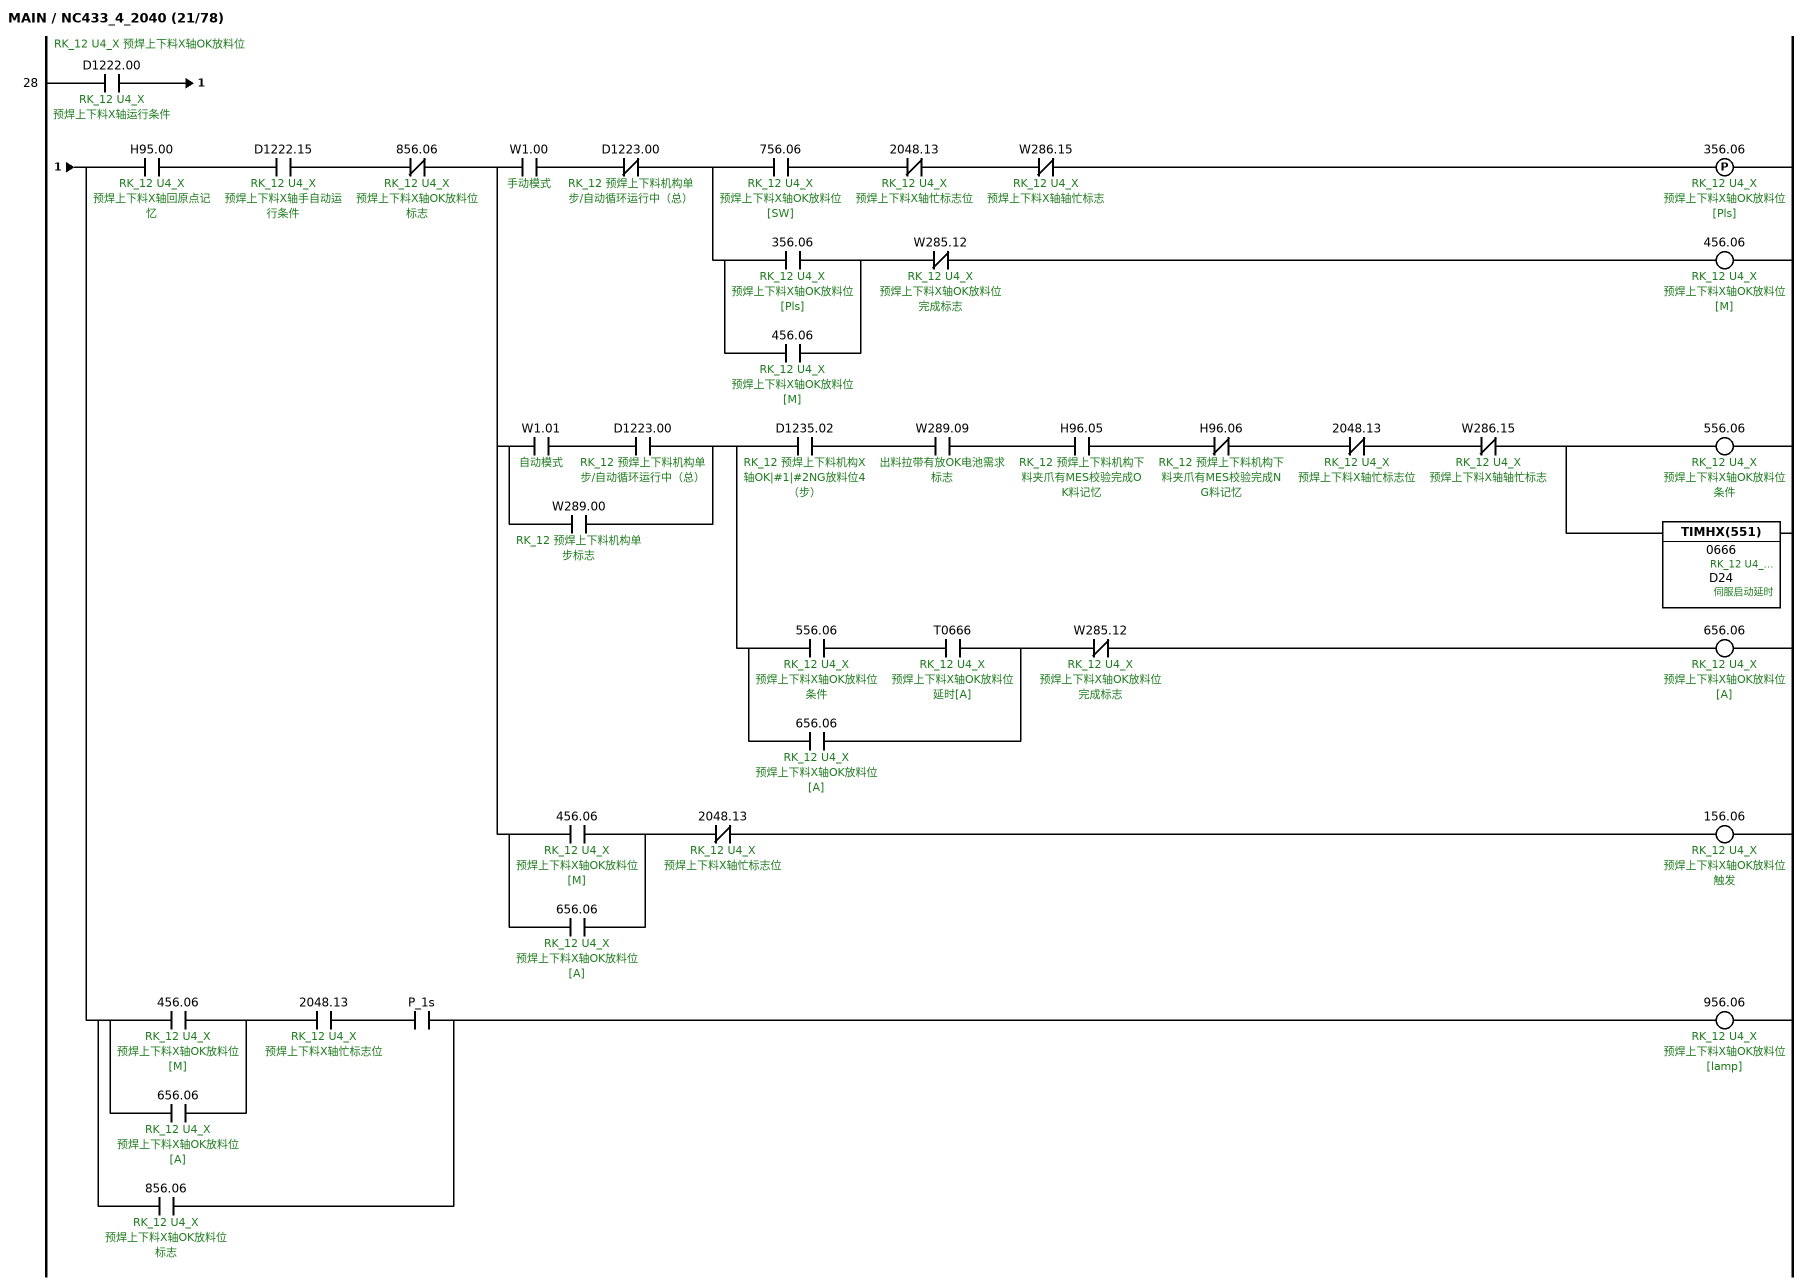
; [picture p168: MAIN / NC433_4_2040, rungs 28-28]
; rung 28: RK_12 U4_X 预焊上下料X轴OK放料位
LD D1222.00  ; RK_12 U4_X 预焊上下料X轴运行条件
OUT TR0
AND H95.00  ; RK_12 U4_X 预焊上下料X轴回原点记忆
AND D1222.15  ; RK_12 U4_X 预焊上下料X轴手自动运行条件
ANDNOT 856.06  ; RK_12 U4_X 预焊上下料X轴OK放料位标志
OUT TR1
AND W1.00  ; 手动模式
ANDNOT D1223.00  ; RK_12 预焊上下料机构单步/自动循环运行中（总）
OUT TR2
AND 756.06  ; RK_12 U4_X 预焊上下料X轴OK放料位[SW]
ANDNOT 2048.13  ; RK_12 U4_X 预焊上下料X轴忙标志位
ANDNOT W286.15  ; RK_12 U4_X 预焊上下料X轴轴忙标志
DIFU(013) 356.06  ; RK_12 U4_X 预焊上下料X轴OK放料位[Pls]
LD TR2
LD 356.06  ; RK_12 U4_X 预焊上下料X轴OK放料位[Pls]
OR 456.06  ; RK_12 U4_X 预焊上下料X轴OK放料位[M]
ANDLD
ANDNOT W285.12  ; RK_12 U4_X 预焊上下料X轴OK放料位完成标志
OUT 456.06  ; RK_12 U4_X 预焊上下料X轴OK放料位[M]
LD TR1
LD W1.01  ; 自动模式
AND D1223.00  ; RK_12 预焊上下料机构单步/自动循环运行中（总）
OR W289.00  ; RK_12 预焊上下料机构单步标志
ANDLD
OUT TR2
AND D1235.02  ; RK_12 预焊上下料机构X轴OK|#1|#2NG放料位4（步）
AND W289.09  ; 出料拉带有放OK电池需求标志
AND H96.05  ; RK_12 预焊上下料机构下料夹爪有MES校验完成OK料记忆
ANDNOT H96.06  ; RK_12 预焊上下料机构下料夹爪有MES校验完成NG料记忆
ANDNOT 2048.13  ; RK_12 U4_X 预焊上下料X轴忙标志位
ANDNOT W286.15  ; RK_12 U4_X 预焊上下料X轴轴忙标志
OUT 556.06  ; RK_12 U4_X 预焊上下料X轴OK放料位条件
TIMHX(551) 0666 D24  ; 伺服启动延时, RK_12 U4_X 预焊上下料X轴OK放料位延时[A]
LD TR2
LD 556.06  ; RK_12 U4_X 预焊上下料X轴OK放料位条件
AND T0666  ; RK_12 U4_X 预焊上下料X轴OK放料位延时[A]
OR 656.06  ; RK_12 U4_X 预焊上下料X轴OK放料位[A]
ANDLD
ANDNOT W285.12  ; RK_12 U4_X 预焊上下料X轴OK放料位完成标志
OUT 656.06  ; RK_12 U4_X 预焊上下料X轴OK放料位[A]
LD TR1
LD 456.06  ; RK_12 U4_X 预焊上下料X轴OK放料位[M]
OR 656.06  ; RK_12 U4_X 预焊上下料X轴OK放料位[A]
ANDLD
ANDNOT 2048.13  ; RK_12 U4_X 预焊上下料X轴忙标志位
OUT 156.06  ; RK_12 U4_X 预焊上下料X轴OK放料位触发
LD TR0
LD 456.06  ; RK_12 U4_X 预焊上下料X轴OK放料位[M]
OR 656.06  ; RK_12 U4_X 预焊上下料X轴OK放料位[A]
AND 2048.13  ; RK_12 U4_X 预焊上下料X轴忙标志位
AND P_1s
OR 856.06  ; RK_12 U4_X 预焊上下料X轴OK放料位标志
ANDLD
OUT 956.06  ; RK_12 U4_X 预焊上下料X轴OK放料位[lamp]

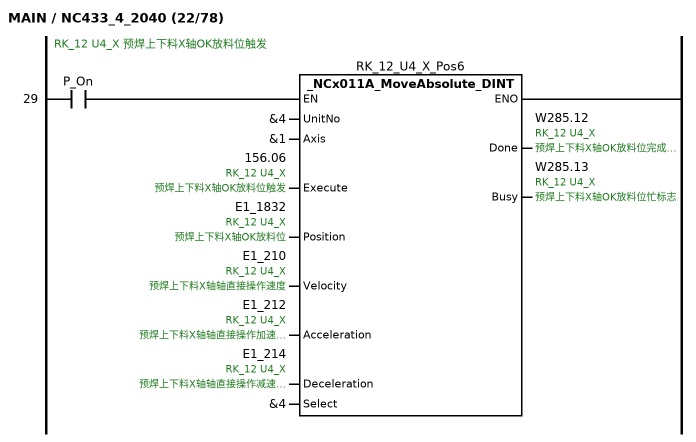
; rung 29: RK_12 U4_X 预焊上下料X轴OK放料位触发
LD P_On
CALL RK_12_U4_X_Pos6 : _NCx011A_MoveAbsolute_DINT (UnitNo := &4, Axis := &1, Execute := 156.06, Position := E1_1832, Velocity := E1_210, Acceleration := E1_212, Deceleration := E1_214, Select := &4, Done => W285.12, Busy => W285.13)  ; RK_12 U4_X 预焊上下料X轴OK放料位触发, RK_12 U4_X 预焊上下料X轴OK放料位, RK_12 U4_X 预焊上下料X轴轴直接操作速度, RK_12 U4_X 预焊上下料X轴轴直接操作加速时间, RK_12 U4_X 预焊上下料X轴轴直接操作减速时间, RK_12 U4_X 预焊上下料X轴OK放料位完成标志, RK_12 U4_X 预焊上下料X轴OK放料位忙标志

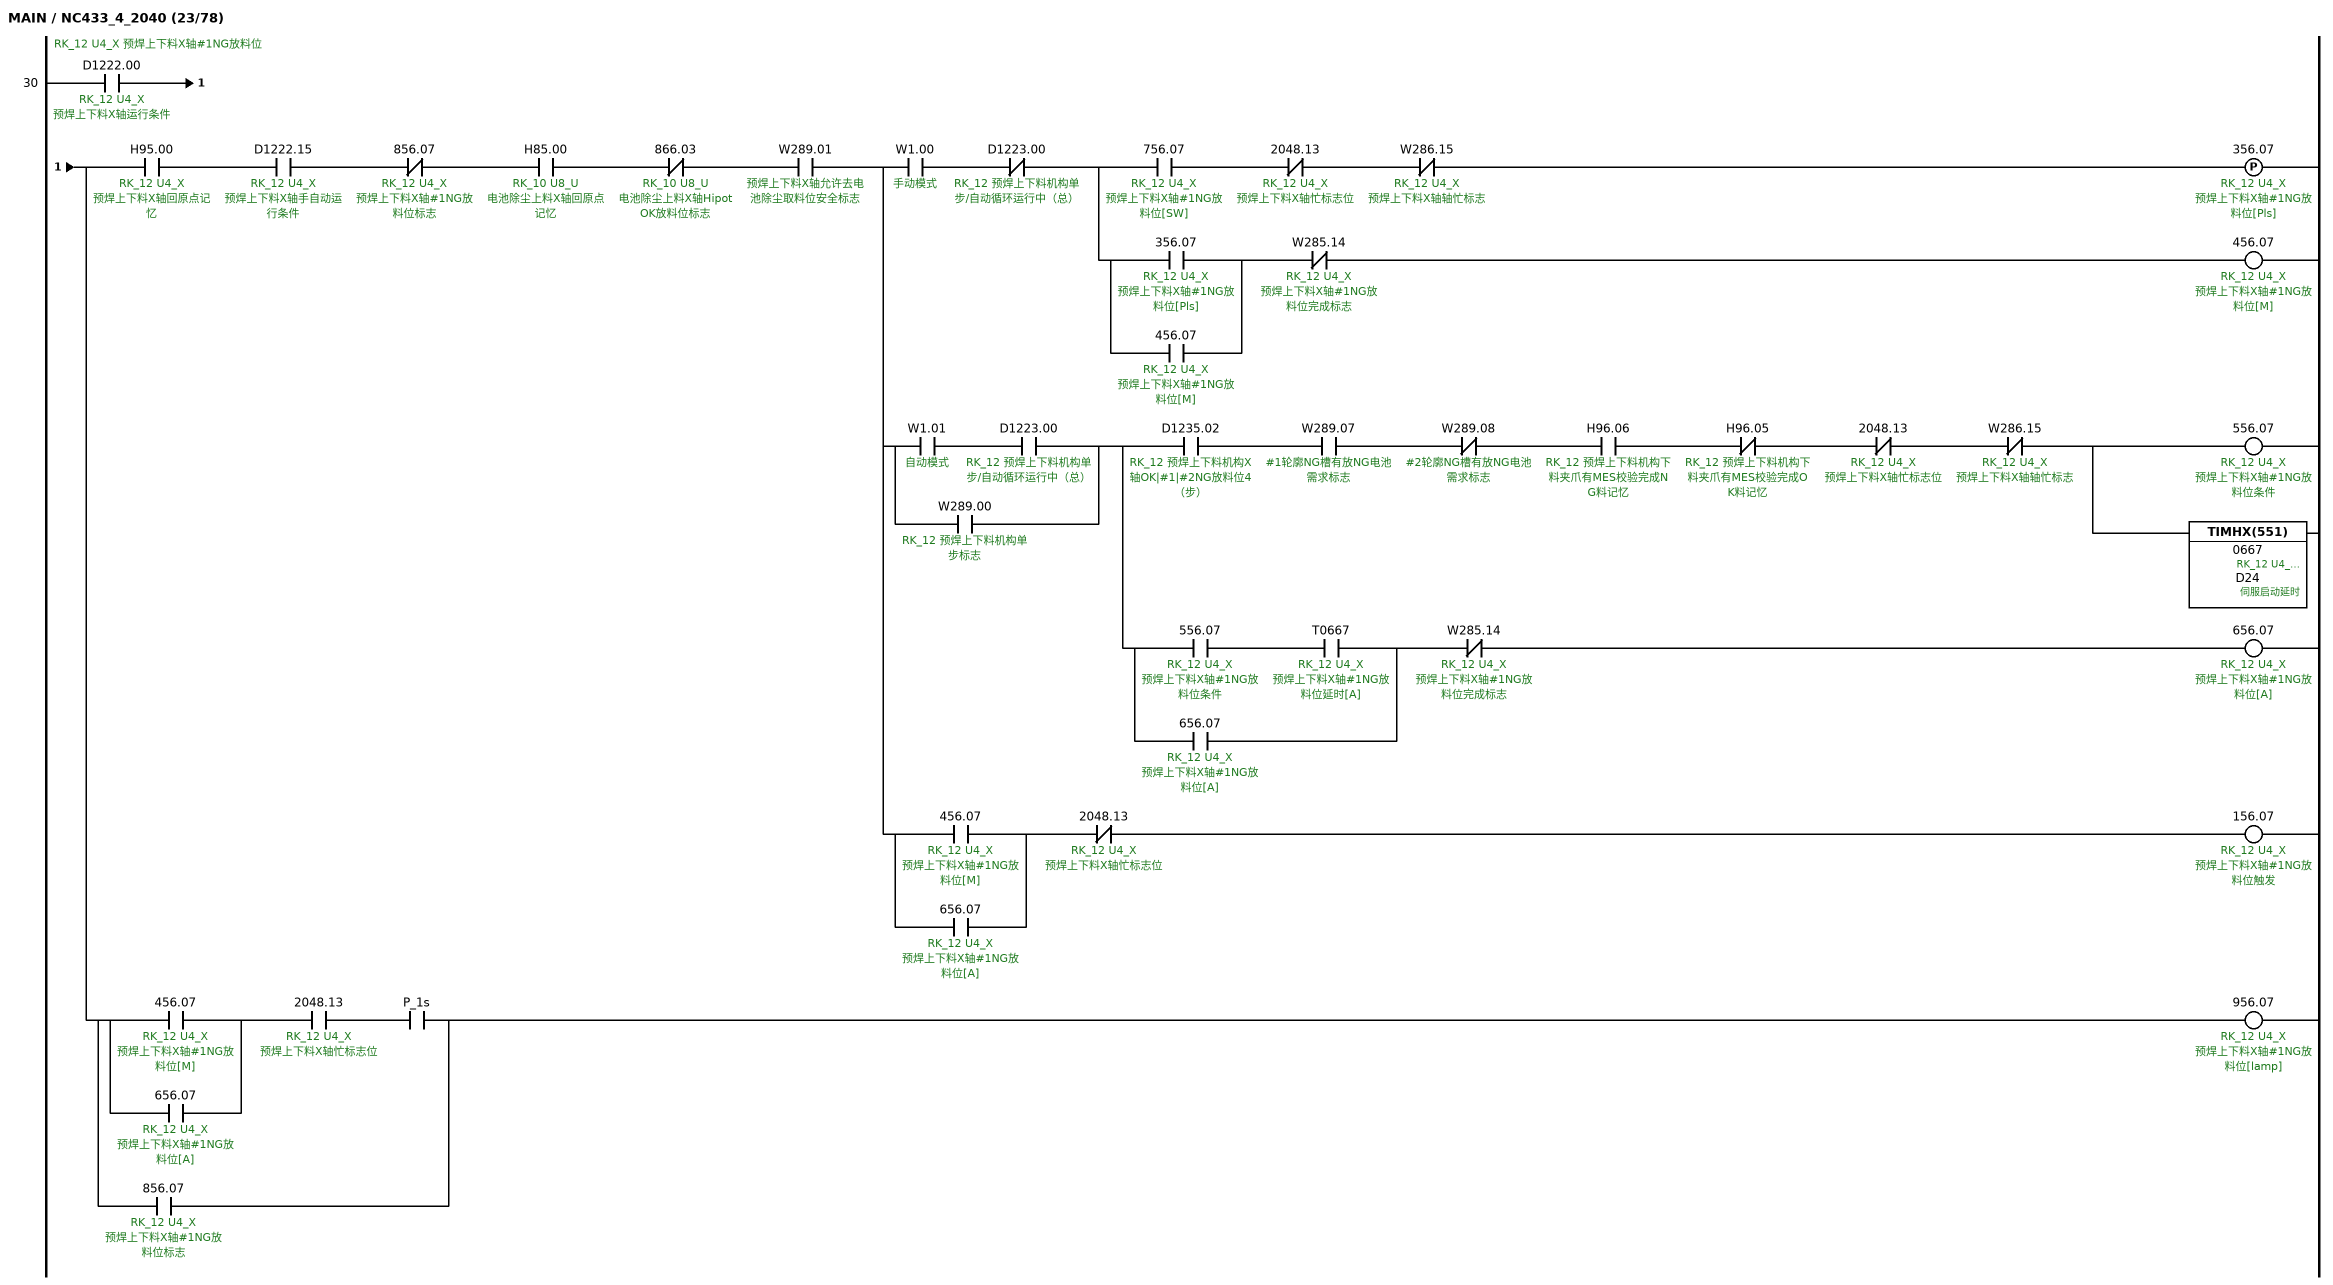
; rung 30: RK_12 U4_X 预焊上下料X轴#1NG放料位
LD D1222.00  ; RK_12 U4_X 预焊上下料X轴运行条件
OUT TR0
AND H95.00  ; RK_12 U4_X 预焊上下料X轴回原点记忆
AND D1222.15  ; RK_12 U4_X 预焊上下料X轴手自动运行条件
ANDNOT 856.07  ; RK_12 U4_X 预焊上下料X轴#1NG放料位标志
AND H85.00  ; RK_10 U8_U 电池除尘上料X轴回原点记忆
ANDNOT 866.03  ; RK_10 U8_U 电池除尘上料X轴Hipot OK放料位标志
AND W289.01  ; 预焊上下料X轴允许去电池除尘取料位安全标志
OUT TR1
AND W1.00  ; 手动模式
ANDNOT D1223.00  ; RK_12 预焊上下料机构单步/自动循环运行中（总）
OUT TR2
AND 756.07  ; RK_12 U4_X 预焊上下料X轴#1NG放料位[SW]
ANDNOT 2048.13  ; RK_12 U4_X 预焊上下料X轴忙标志位
ANDNOT W286.15  ; RK_12 U4_X 预焊上下料X轴轴忙标志
DIFU(013) 356.07  ; RK_12 U4_X 预焊上下料X轴#1NG放料位[Pls]
LD TR2
LD 356.07  ; RK_12 U4_X 预焊上下料X轴#1NG放料位[Pls]
OR 456.07  ; RK_12 U4_X 预焊上下料X轴#1NG放料位[M]
ANDLD
ANDNOT W285.14  ; RK_12 U4_X 预焊上下料X轴#1NG放料位完成标志
OUT 456.07  ; RK_12 U4_X 预焊上下料X轴#1NG放料位[M]
LD TR1
LD W1.01  ; 自动模式
AND D1223.00  ; RK_12 预焊上下料机构单步/自动循环运行中（总）
OR W289.00  ; RK_12 预焊上下料机构单步标志
ANDLD
OUT TR2
AND D1235.02  ; RK_12 预焊上下料机构X轴OK|#1|#2NG放料位4（步）
AND W289.07  ; #1轮廓NG槽有放NG电池需求标志
ANDNOT W289.08  ; #2轮廓NG槽有放NG电池需求标志
AND H96.06  ; RK_12 预焊上下料机构下料夹爪有MES校验完成NG料记忆
ANDNOT H96.05  ; RK_12 预焊上下料机构下料夹爪有MES校验完成OK料记忆
ANDNOT 2048.13  ; RK_12 U4_X 预焊上下料X轴忙标志位
ANDNOT W286.15  ; RK_12 U4_X 预焊上下料X轴轴忙标志
OUT 556.07  ; RK_12 U4_X 预焊上下料X轴#1NG放料位条件
TIMHX(551) 0667 D24  ; 伺服启动延时, RK_12 U4_X 预焊上下料X轴#1NG放料位延时[A]
LD TR2
LD 556.07  ; RK_12 U4_X 预焊上下料X轴#1NG放料位条件
AND T0667  ; RK_12 U4_X 预焊上下料X轴#1NG放料位延时[A]
OR 656.07  ; RK_12 U4_X 预焊上下料X轴#1NG放料位[A]
ANDLD
ANDNOT W285.14  ; RK_12 U4_X 预焊上下料X轴#1NG放料位完成标志
OUT 656.07  ; RK_12 U4_X 预焊上下料X轴#1NG放料位[A]
LD TR1
LD 456.07  ; RK_12 U4_X 预焊上下料X轴#1NG放料位[M]
OR 656.07  ; RK_12 U4_X 预焊上下料X轴#1NG放料位[A]
ANDLD
ANDNOT 2048.13  ; RK_12 U4_X 预焊上下料X轴忙标志位
OUT 156.07  ; RK_12 U4_X 预焊上下料X轴#1NG放料位触发
LD TR0
LD 456.07  ; RK_12 U4_X 预焊上下料X轴#1NG放料位[M]
OR 656.07  ; RK_12 U4_X 预焊上下料X轴#1NG放料位[A]
AND 2048.13  ; RK_12 U4_X 预焊上下料X轴忙标志位
AND P_1s
OR 856.07  ; RK_12 U4_X 预焊上下料X轴#1NG放料位标志
ANDLD
OUT 956.07  ; RK_12 U4_X 预焊上下料X轴#1NG放料位[lamp]

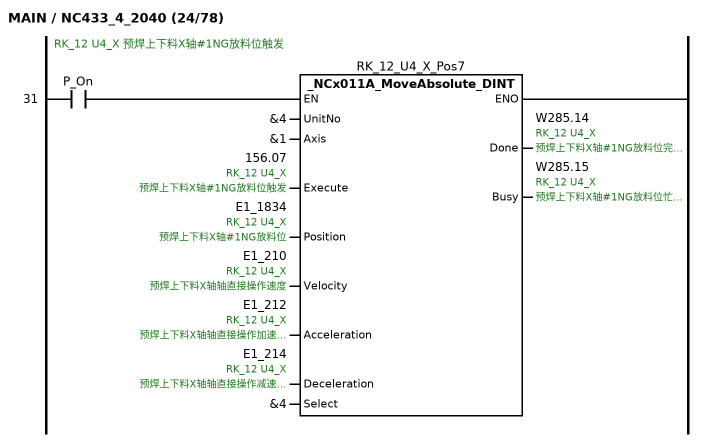
; rung 31: RK_12 U4_X 预焊上下料X轴#1NG放料位触发
LD P_On
CALL RK_12_U4_X_Pos7 : _NCx011A_MoveAbsolute_DINT (UnitNo := &4, Axis := &1, Execute := 156.07, Position := E1_1834, Velocity := E1_210, Acceleration := E1_212, Deceleration := E1_214, Select := &4, Done => W285.14, Busy => W285.15)  ; RK_12 U4_X 预焊上下料X轴#1NG放料位触发, RK_12 U4_X 预焊上下料X轴#1NG放料位, RK_12 U4_X 预焊上下料X轴轴直接操作速度, RK_12 U4_X 预焊上下料X轴轴直接操作加速时间, RK_12 U4_X 预焊上下料X轴轴直接操作减速时间, RK_12 U4_X 预焊上下料X轴#1NG放料位完成标志, RK_12 U4_X 预焊上下料X轴#1NG放料位忙标志

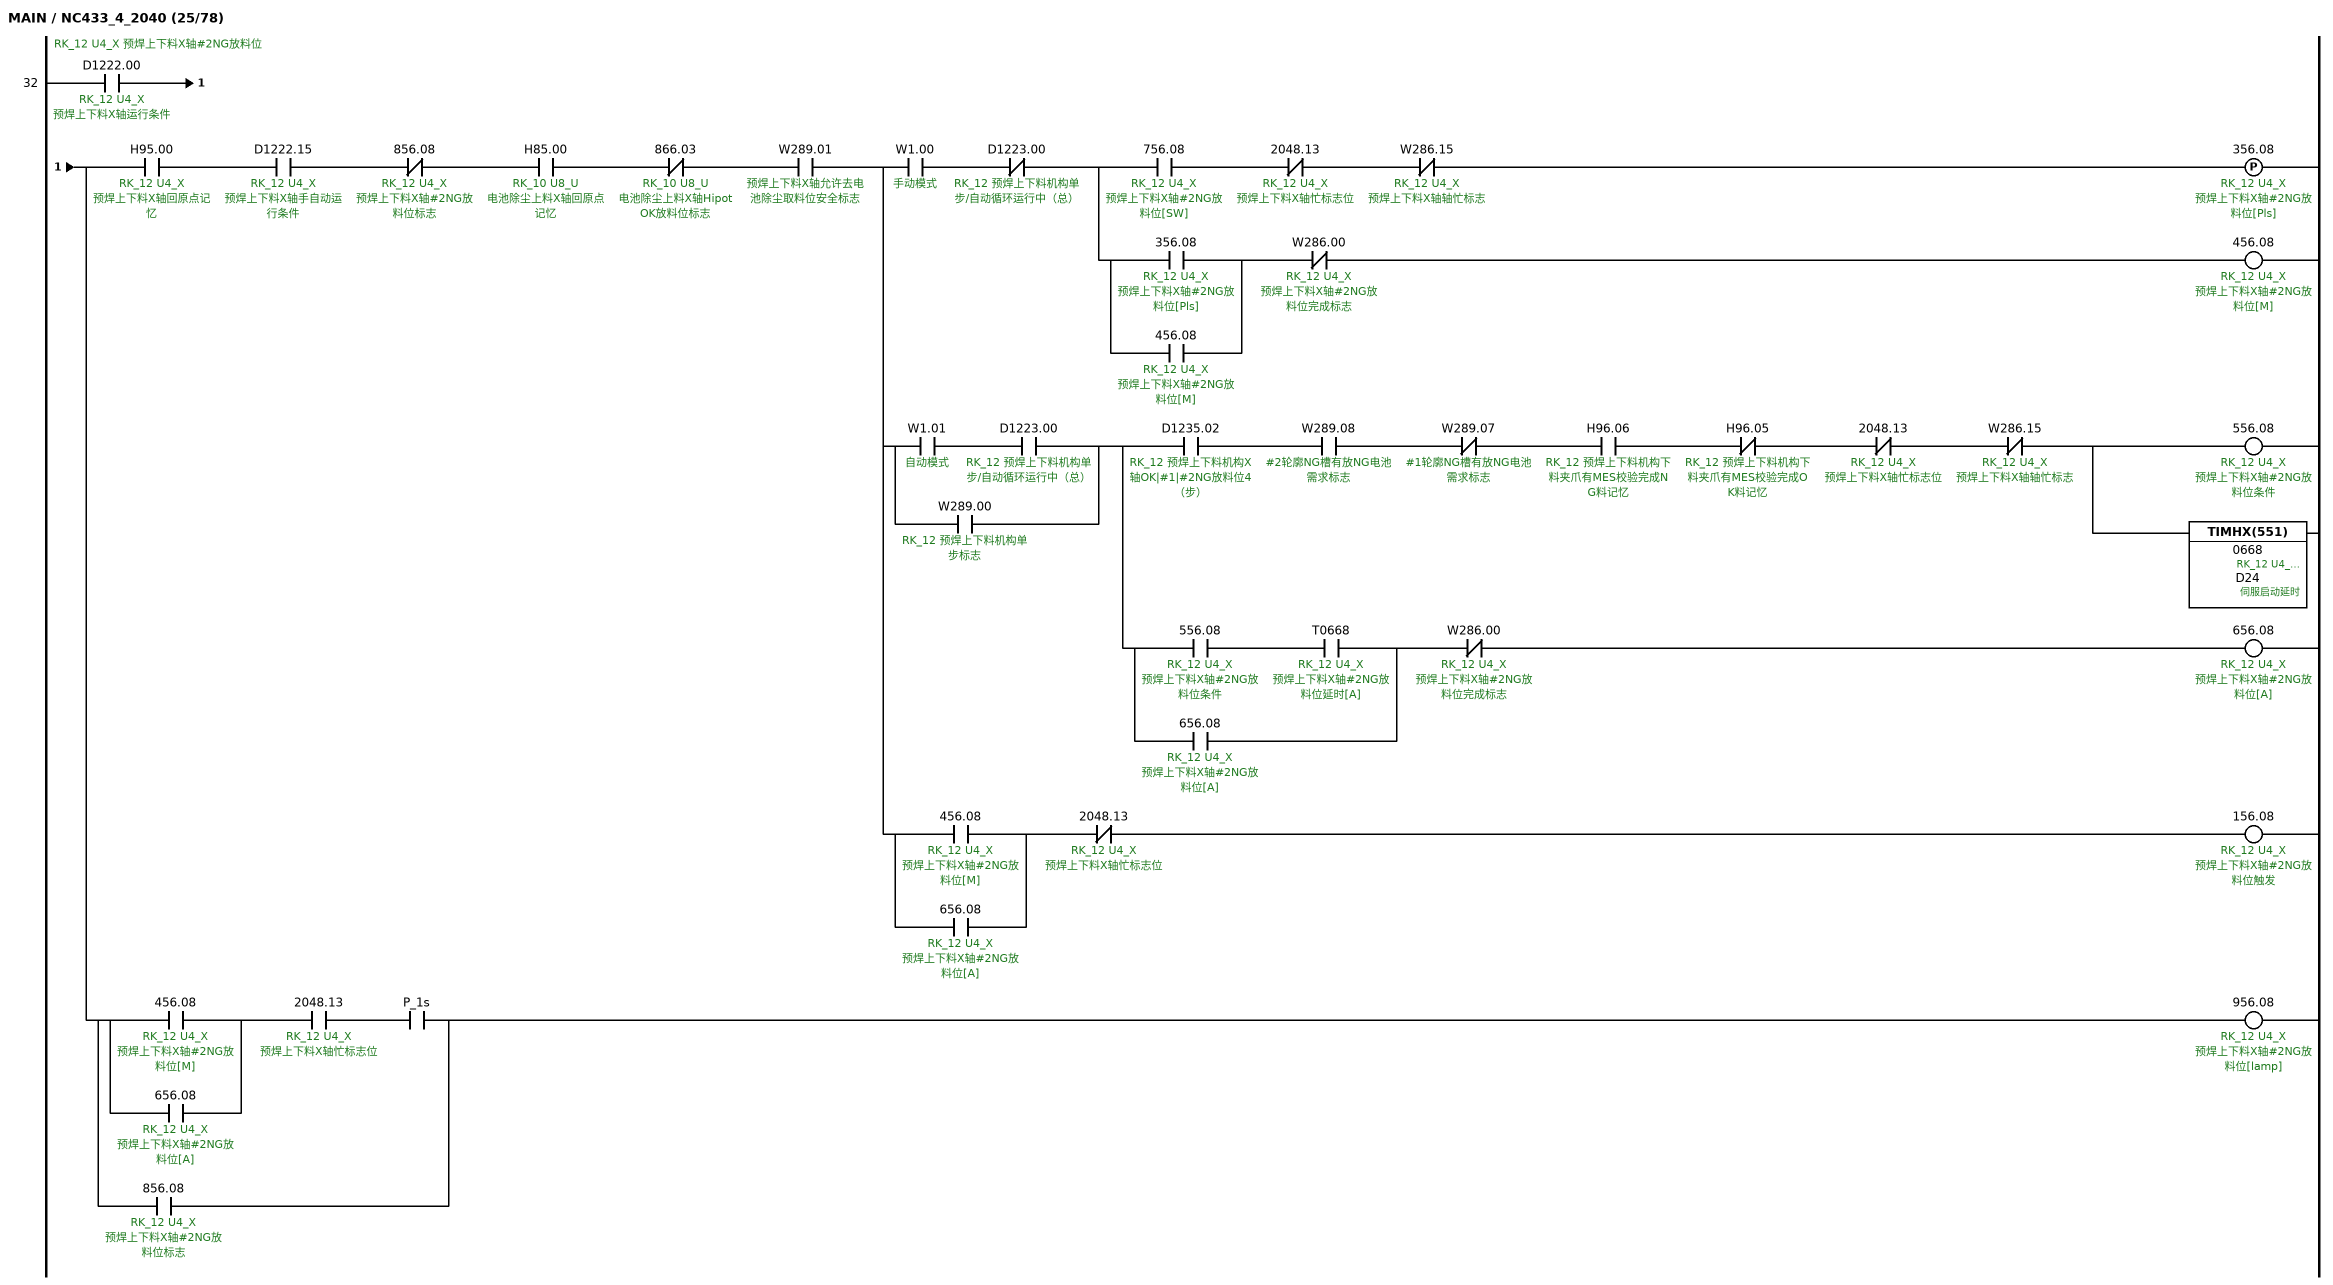
; rung 32: RK_12 U4_X 预焊上下料X轴#2NG放料位
LD D1222.00  ; RK_12 U4_X 预焊上下料X轴运行条件
OUT TR0
AND H95.00  ; RK_12 U4_X 预焊上下料X轴回原点记忆
AND D1222.15  ; RK_12 U4_X 预焊上下料X轴手自动运行条件
ANDNOT 856.08  ; RK_12 U4_X 预焊上下料X轴#2NG放料位标志
AND H85.00  ; RK_10 U8_U 电池除尘上料X轴回原点记忆
ANDNOT 866.03  ; RK_10 U8_U 电池除尘上料X轴Hipot OK放料位标志
AND W289.01  ; 预焊上下料X轴允许去电池除尘取料位安全标志
OUT TR1
AND W1.00  ; 手动模式
ANDNOT D1223.00  ; RK_12 预焊上下料机构单步/自动循环运行中（总）
OUT TR2
AND 756.08  ; RK_12 U4_X 预焊上下料X轴#2NG放料位[SW]
ANDNOT 2048.13  ; RK_12 U4_X 预焊上下料X轴忙标志位
ANDNOT W286.15  ; RK_12 U4_X 预焊上下料X轴轴忙标志
DIFU(013) 356.08  ; RK_12 U4_X 预焊上下料X轴#2NG放料位[Pls]
LD TR2
LD 356.08  ; RK_12 U4_X 预焊上下料X轴#2NG放料位[Pls]
OR 456.08  ; RK_12 U4_X 预焊上下料X轴#2NG放料位[M]
ANDLD
ANDNOT W286.00  ; RK_12 U4_X 预焊上下料X轴#2NG放料位完成标志
OUT 456.08  ; RK_12 U4_X 预焊上下料X轴#2NG放料位[M]
LD TR1
LD W1.01  ; 自动模式
AND D1223.00  ; RK_12 预焊上下料机构单步/自动循环运行中（总）
OR W289.00  ; RK_12 预焊上下料机构单步标志
ANDLD
OUT TR2
AND D1235.02  ; RK_12 预焊上下料机构X轴OK|#1|#2NG放料位4（步）
AND W289.08  ; #2轮廓NG槽有放NG电池需求标志
ANDNOT W289.07  ; #1轮廓NG槽有放NG电池需求标志
AND H96.06  ; RK_12 预焊上下料机构下料夹爪有MES校验完成NG料记忆
ANDNOT H96.05  ; RK_12 预焊上下料机构下料夹爪有MES校验完成OK料记忆
ANDNOT 2048.13  ; RK_12 U4_X 预焊上下料X轴忙标志位
ANDNOT W286.15  ; RK_12 U4_X 预焊上下料X轴轴忙标志
OUT 556.08  ; RK_12 U4_X 预焊上下料X轴#2NG放料位条件
TIMHX(551) 0668 D24  ; 伺服启动延时, RK_12 U4_X 预焊上下料X轴#2NG放料位延时[A]
LD TR2
LD 556.08  ; RK_12 U4_X 预焊上下料X轴#2NG放料位条件
AND T0668  ; RK_12 U4_X 预焊上下料X轴#2NG放料位延时[A]
OR 656.08  ; RK_12 U4_X 预焊上下料X轴#2NG放料位[A]
ANDLD
ANDNOT W286.00  ; RK_12 U4_X 预焊上下料X轴#2NG放料位完成标志
OUT 656.08  ; RK_12 U4_X 预焊上下料X轴#2NG放料位[A]
LD TR1
LD 456.08  ; RK_12 U4_X 预焊上下料X轴#2NG放料位[M]
OR 656.08  ; RK_12 U4_X 预焊上下料X轴#2NG放料位[A]
ANDLD
ANDNOT 2048.13  ; RK_12 U4_X 预焊上下料X轴忙标志位
OUT 156.08  ; RK_12 U4_X 预焊上下料X轴#2NG放料位触发
LD TR0
LD 456.08  ; RK_12 U4_X 预焊上下料X轴#2NG放料位[M]
OR 656.08  ; RK_12 U4_X 预焊上下料X轴#2NG放料位[A]
AND 2048.13  ; RK_12 U4_X 预焊上下料X轴忙标志位
AND P_1s
OR 856.08  ; RK_12 U4_X 预焊上下料X轴#2NG放料位标志
ANDLD
OUT 956.08  ; RK_12 U4_X 预焊上下料X轴#2NG放料位[lamp]

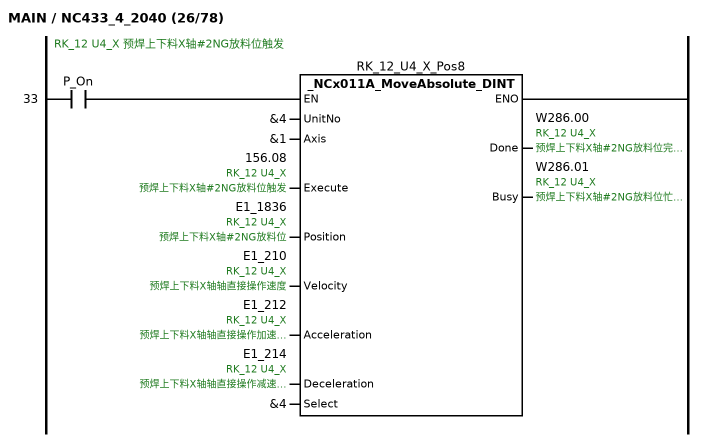
; rung 33: RK_12 U4_X 预焊上下料X轴#2NG放料位触发
LD P_On
CALL RK_12_U4_X_Pos8 : _NCx011A_MoveAbsolute_DINT (UnitNo := &4, Axis := &1, Execute := 156.08, Position := E1_1836, Velocity := E1_210, Acceleration := E1_212, Deceleration := E1_214, Select := &4, Done => W286.00, Busy => W286.01)  ; RK_12 U4_X 预焊上下料X轴#2NG放料位触发, RK_12 U4_X 预焊上下料X轴#2NG放料位, RK_12 U4_X 预焊上下料X轴轴直接操作速度, RK_12 U4_X 预焊上下料X轴轴直接操作加速时间, RK_12 U4_X 预焊上下料X轴轴直接操作减速时间, RK_12 U4_X 预焊上下料X轴#2NG放料位完成标志, RK_12 U4_X 预焊上下料X轴#2NG放料位忙标志

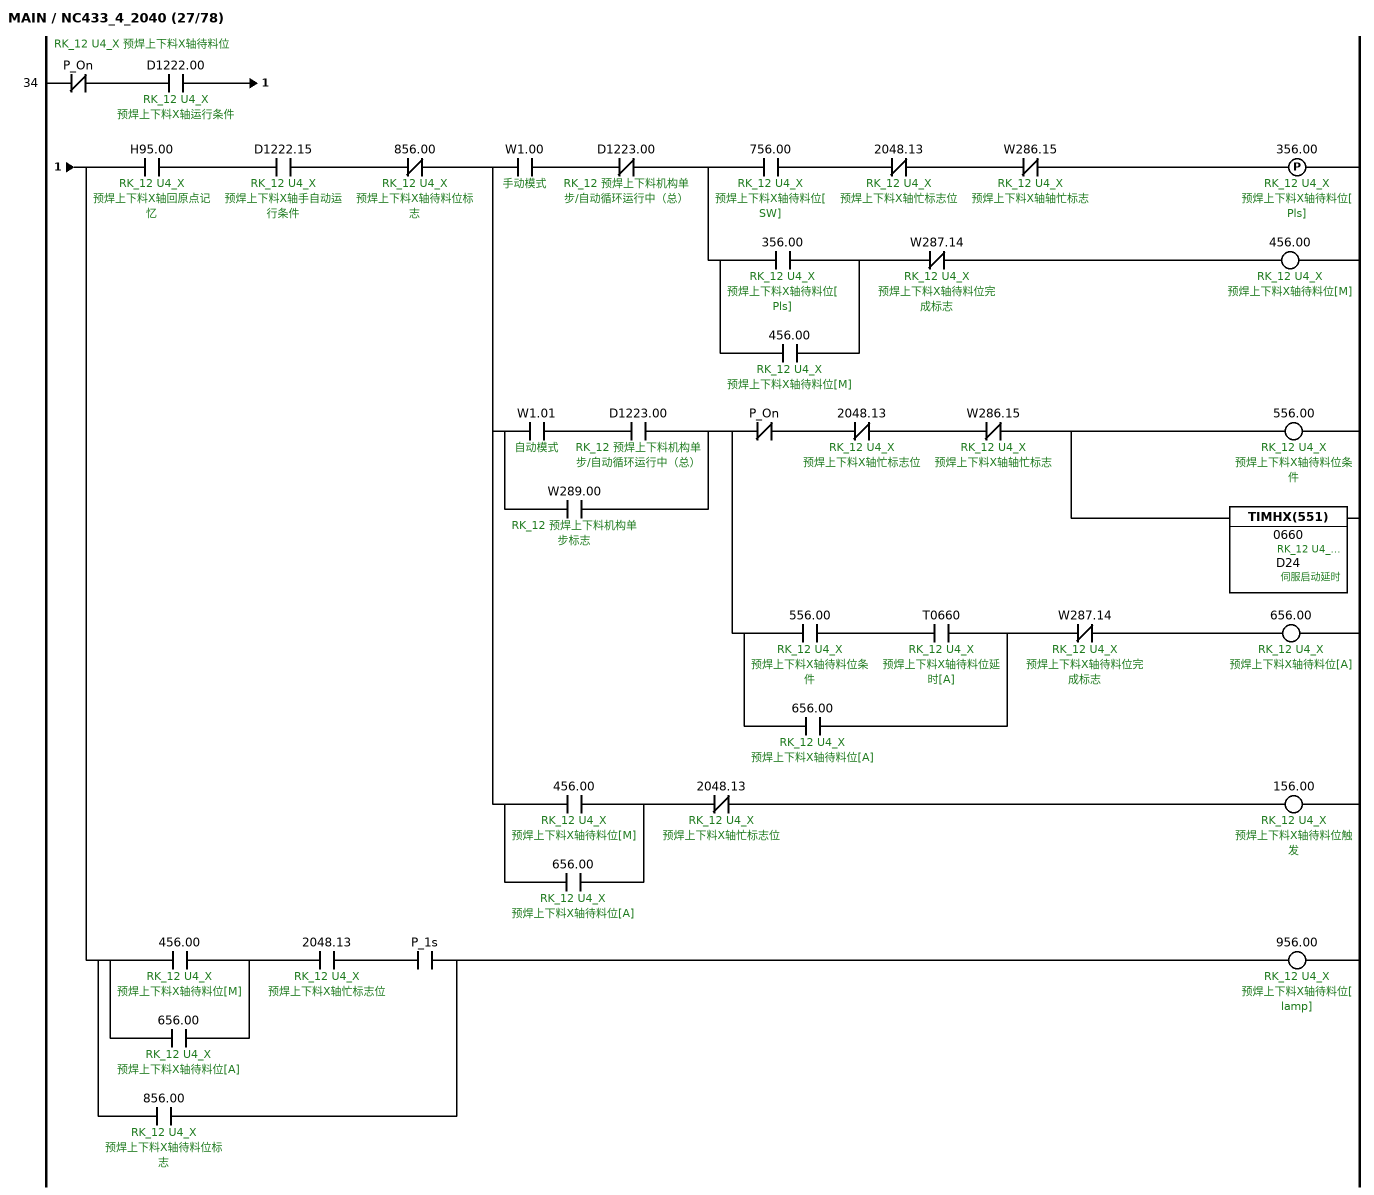
; rung 34: RK_12 U4_X 预焊上下料X轴待料位
LDNOT P_On
AND D1222.00  ; RK_12 U4_X 预焊上下料X轴运行条件
OUT TR0
AND H95.00  ; RK_12 U4_X 预焊上下料X轴回原点记忆
AND D1222.15  ; RK_12 U4_X 预焊上下料X轴手自动运行条件
ANDNOT 856.00  ; RK_12 U4_X 预焊上下料X轴待料位标志
OUT TR1
AND W1.00  ; 手动模式
ANDNOT D1223.00  ; RK_12 预焊上下料机构单步/自动循环运行中（总）
OUT TR2
AND 756.00  ; RK_12 U4_X 预焊上下料X轴待料位[SW]
ANDNOT 2048.13  ; RK_12 U4_X 预焊上下料X轴忙标志位
ANDNOT W286.15  ; RK_12 U4_X 预焊上下料X轴轴忙标志
DIFU(013) 356.00  ; RK_12 U4_X 预焊上下料X轴待料位[Pls]
LD TR2
LD 356.00  ; RK_12 U4_X 预焊上下料X轴待料位[Pls]
OR 456.00  ; RK_12 U4_X 预焊上下料X轴待料位[M]
ANDLD
ANDNOT W287.14  ; RK_12 U4_X 预焊上下料X轴待料位完成标志
OUT 456.00  ; RK_12 U4_X 预焊上下料X轴待料位[M]
LD TR1
LD W1.01  ; 自动模式
AND D1223.00  ; RK_12 预焊上下料机构单步/自动循环运行中（总）
OR W289.00  ; RK_12 预焊上下料机构单步标志
ANDLD
OUT TR2
ANDNOT P_On  // RK_12 U4_X 预焊上下料X轴待料位（步）
ANDNOT 2048.13  ; RK_12 U4_X 预焊上下料X轴忙标志位
ANDNOT W286.15  ; RK_12 U4_X 预焊上下料X轴轴忙标志
OUT 556.00  ; RK_12 U4_X 预焊上下料X轴待料位条件
TIMHX(551) 0660 D24  ; 伺服启动延时, RK_12 U4_X 预焊上下料X轴待料位延时[A]
LD TR2
LD 556.00  ; RK_12 U4_X 预焊上下料X轴待料位条件
AND T0660  ; RK_12 U4_X 预焊上下料X轴待料位延时[A]
OR 656.00  ; RK_12 U4_X 预焊上下料X轴待料位[A]
ANDLD
ANDNOT W287.14  ; RK_12 U4_X 预焊上下料X轴待料位完成标志
OUT 656.00  ; RK_12 U4_X 预焊上下料X轴待料位[A]
LD TR1
LD 456.00  ; RK_12 U4_X 预焊上下料X轴待料位[M]
OR 656.00  ; RK_12 U4_X 预焊上下料X轴待料位[A]
ANDLD
ANDNOT 2048.13  ; RK_12 U4_X 预焊上下料X轴忙标志位
OUT 156.00  ; RK_12 U4_X 预焊上下料X轴待料位触发
LD TR0
LD 456.00  ; RK_12 U4_X 预焊上下料X轴待料位[M]
OR 656.00  ; RK_12 U4_X 预焊上下料X轴待料位[A]
AND 2048.13  ; RK_12 U4_X 预焊上下料X轴忙标志位
AND P_1s
OR 856.00  ; RK_12 U4_X 预焊上下料X轴待料位标志
ANDLD
OUT 956.00  ; RK_12 U4_X 预焊上下料X轴待料位[lamp]

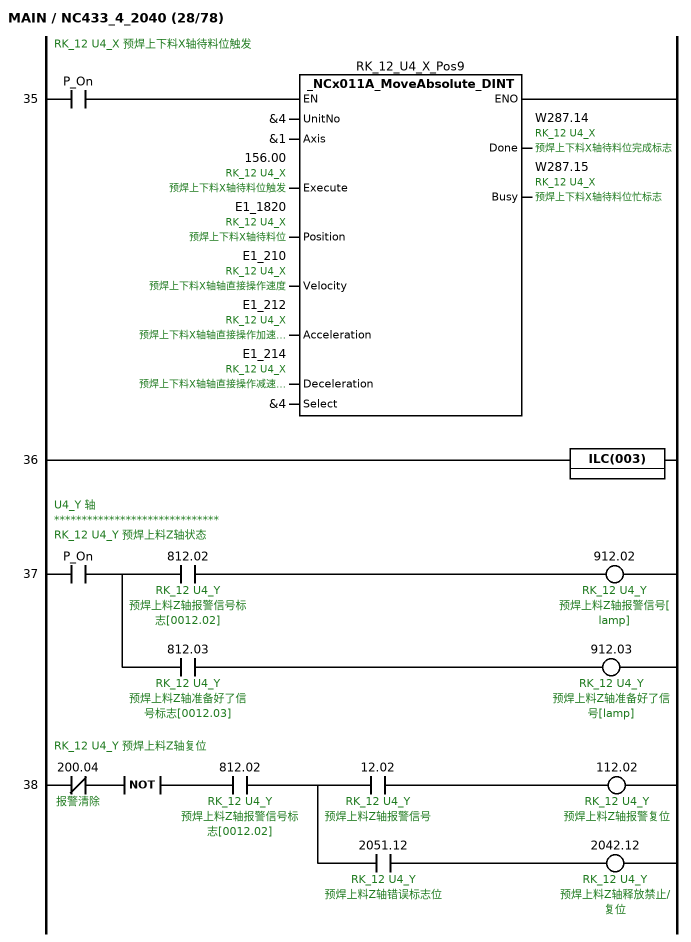
; rung 35: RK_12 U4_X 预焊上下料X轴待料位触发
LD P_On
CALL RK_12_U4_X_Pos9 : _NCx011A_MoveAbsolute_DINT (UnitNo := &4, Axis := &1, Execute := 156.00, Position := E1_1820, Velocity := E1_210, Acceleration := E1_212, Deceleration := E1_214, Select := &4, Done => W287.14, Busy => W287.15)  ; RK_12 U4_X 预焊上下料X轴待料位触发, RK_12 U4_X 预焊上下料X轴待料位, RK_12 U4_X 预焊上下料X轴轴直接操作速度, RK_12 U4_X 预焊上下料X轴轴直接操作加速时间, RK_12 U4_X 预焊上下料X轴轴直接操作减速时间, RK_12 U4_X 预焊上下料X轴待料位完成标志, RK_12 U4_X 预焊上下料X轴待料位忙标志
; rung 36
ILC(003)
; rung 37: U4_Y 轴 / ****************************** / RK_12 U4_Y 预焊上料Z轴状态
LD P_On
OUT TR0
AND 812.02  ; RK_12 U4_Y 预焊上料Z轴报警信号标志[0012.02]
OUT 912.02  ; RK_12 U4_Y 预焊上料Z轴报警信号[lamp]
LD TR0
AND 812.03  ; RK_12 U4_Y 预焊上料Z轴准备好了信号标志[0012.03]
OUT 912.03  ; RK_12 U4_Y 预焊上料Z轴准备好了信号[lamp]
; rung 38: RK_12 U4_Y 预焊上料Z轴复位
LDNOT 200.04  ; 报警清除
NOT(520)
AND 812.02  ; RK_12 U4_Y 预焊上料Z轴报警信号标志[0012.02]
OUT TR0
AND 12.02  ; RK_12 U4_Y 预焊上料Z轴报警信号
OUT 112.02  ; RK_12 U4_Y 预焊上料Z轴报警复位
LD TR0
AND 2051.12  ; RK_12 U4_Y 预焊上料Z轴错误标志位
OUT 2042.12  ; RK_12 U4_Y 预焊上料Z轴释放禁止/复位

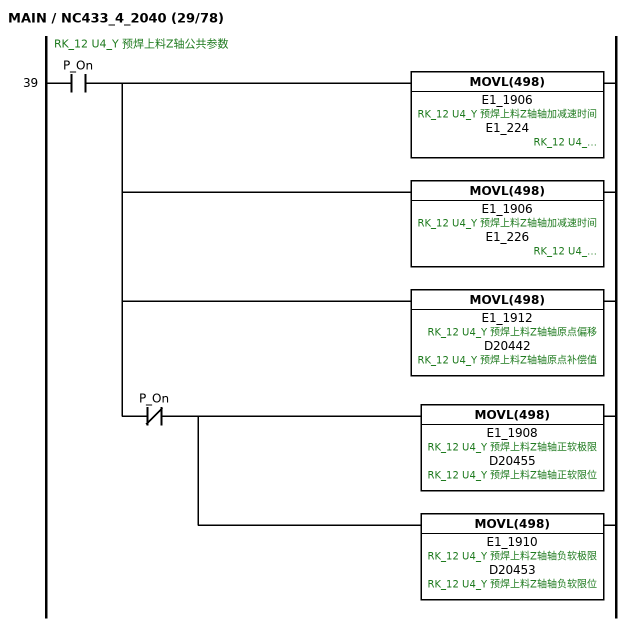
; rung 39: RK_12 U4_Y 预焊上料Z轴公共参数
LD P_On
MOVL(498) E1_1906 E1_224  ; RK_12 U4_Y 预焊上料Z轴轴加减速时间, RK_12 U4_Y 预焊上料Z轴轴直接操作加速时间
MOVL(498) E1_1906 E1_226  ; RK_12 U4_Y 预焊上料Z轴轴加减速时间, RK_12 U4_Y 预焊上料Z轴轴直接操作减速时间
MOVL(498) E1_1912 D20442  ; RK_12 U4_Y 预焊上料Z轴轴原点偏移, RK_12 U4_Y 预焊上料Z轴轴原点补偿值
ANDNOT P_On
MOVL(498) E1_1908 D20455  ; RK_12 U4_Y 预焊上料Z轴轴正软极限, RK_12 U4_Y 预焊上料Z轴轴正软限位
MOVL(498) E1_1910 D20453  ; RK_12 U4_Y 预焊上料Z轴轴负软极限, RK_12 U4_Y 预焊上料Z轴轴负软限位

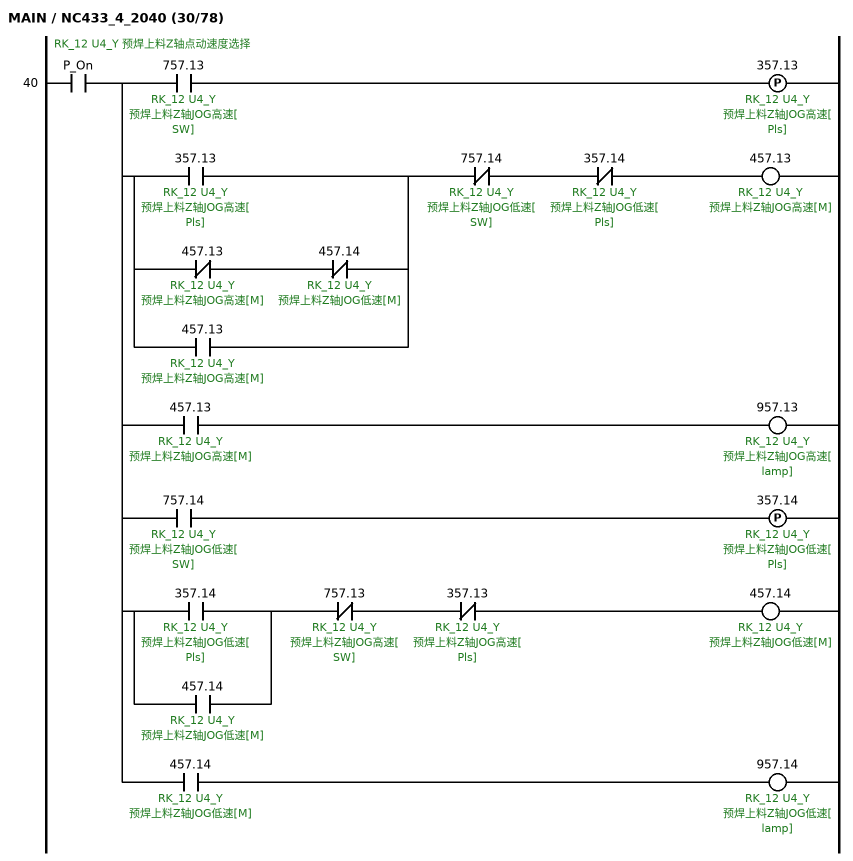
; rung 40: RK_12 U4_Y 预焊上料Z轴点动速度选择
LD P_On
OUT TR0
AND 757.13  ; RK_12 U4_Y 预焊上料Z轴JOG高速[SW]
DIFU(013) 357.13  ; RK_12 U4_Y 预焊上料Z轴JOG高速[Pls]
LD TR0
LD 357.13  ; RK_12 U4_Y 预焊上料Z轴JOG高速[Pls]
LDNOT 457.13  ; RK_12 U4_Y 预焊上料Z轴JOG高速[M]
ANDNOT 457.14  ; RK_12 U4_Y 预焊上料Z轴JOG低速[M]
ORLD
OR 457.13  ; RK_12 U4_Y 预焊上料Z轴JOG高速[M]
ANDLD
ANDNOT 757.14  ; RK_12 U4_Y 预焊上料Z轴JOG低速[SW]
ANDNOT 357.14  ; RK_12 U4_Y 预焊上料Z轴JOG低速[Pls]
OUT 457.13  ; RK_12 U4_Y 预焊上料Z轴JOG高速[M]
LD TR0
AND 457.13  ; RK_12 U4_Y 预焊上料Z轴JOG高速[M]
OUT 957.13  ; RK_12 U4_Y 预焊上料Z轴JOG高速[lamp]
LD TR0
AND 757.14  ; RK_12 U4_Y 预焊上料Z轴JOG低速[SW]
DIFU(013) 357.14  ; RK_12 U4_Y 预焊上料Z轴JOG低速[Pls]
LD TR0
LD 357.14  ; RK_12 U4_Y 预焊上料Z轴JOG低速[Pls]
OR 457.14  ; RK_12 U4_Y 预焊上料Z轴JOG低速[M]
ANDLD
ANDNOT 757.13  ; RK_12 U4_Y 预焊上料Z轴JOG高速[SW]
ANDNOT 357.13  ; RK_12 U4_Y 预焊上料Z轴JOG高速[Pls]
OUT 457.14  ; RK_12 U4_Y 预焊上料Z轴JOG低速[M]
LD TR0
AND 457.14  ; RK_12 U4_Y 预焊上料Z轴JOG低速[M]
OUT 957.14  ; RK_12 U4_Y 预焊上料Z轴JOG低速[lamp]

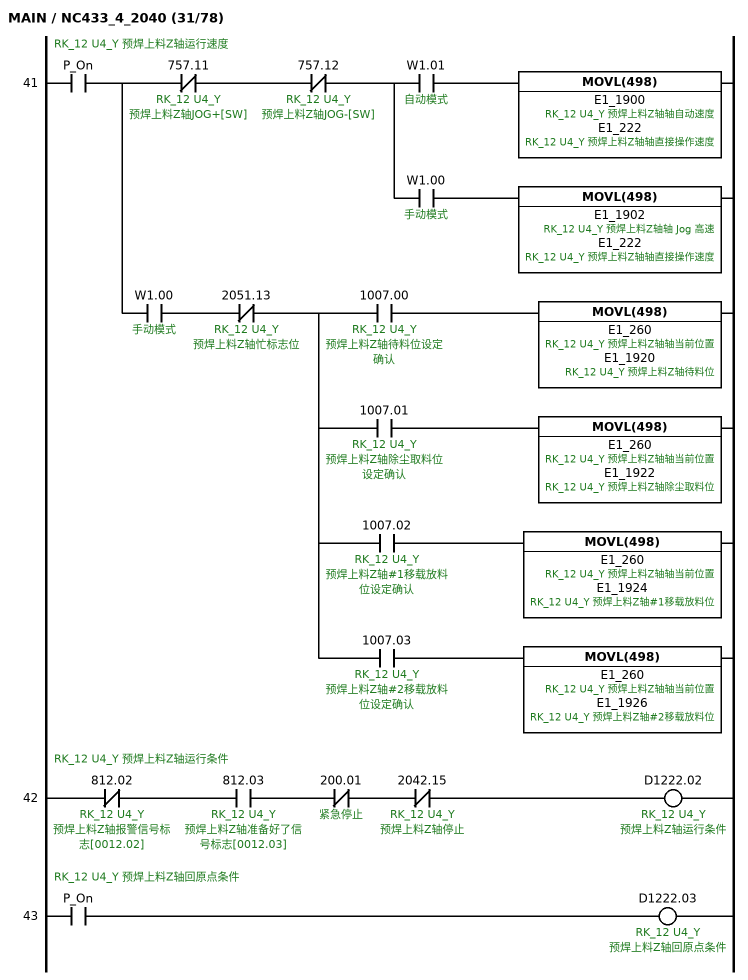
; rung 41: RK_12 U4_Y 预焊上料Z轴运行速度
LD P_On
OUT TR0
ANDNOT 757.11  ; RK_12 U4_Y 预焊上料Z轴JOG+[SW]
ANDNOT 757.12  ; RK_12 U4_Y 预焊上料Z轴JOG-[SW]
OUT TR1
AND W1.01  ; 自动模式
MOVL(498) E1_1900 E1_222  ; RK_12 U4_Y 预焊上料Z轴轴自动速度, RK_12 U4_Y 预焊上料Z轴轴直接操作速度
LD TR1
AND W1.00  ; 手动模式
MOVL(498) E1_1902 E1_222  ; RK_12 U4_Y 预焊上料Z轴轴 Jog 高速, RK_12 U4_Y 预焊上料Z轴轴直接操作速度
LD TR0
AND W1.00  ; 手动模式
ANDNOT 2051.13  ; RK_12 U4_Y 预焊上料Z轴忙标志位
OUT TR0
AND 1007.00  ; RK_12 U4_Y 预焊上料Z轴待料位设定确认
MOVL(498) E1_260 E1_1920  ; RK_12 U4_Y 预焊上料Z轴轴当前位置, RK_12 U4_Y 预焊上料Z轴待料位
LD TR0
AND 1007.01  ; RK_12 U4_Y 预焊上料Z轴除尘取料位设定确认
MOVL(498) E1_260 E1_1922  ; RK_12 U4_Y 预焊上料Z轴轴当前位置, RK_12 U4_Y 预焊上料Z轴除尘取料位
LD TR0
AND 1007.02  ; RK_12 U4_Y 预焊上料Z轴#1移载放料位设定确认
MOVL(498) E1_260 E1_1924  ; RK_12 U4_Y 预焊上料Z轴轴当前位置, RK_12 U4_Y 预焊上料Z轴#1移载放料位
LD TR0
AND 1007.03  ; RK_12 U4_Y 预焊上料Z轴#2移载放料位设定确认
MOVL(498) E1_260 E1_1926  ; RK_12 U4_Y 预焊上料Z轴轴当前位置, RK_12 U4_Y 预焊上料Z轴#2移载放料位
; rung 42: RK_12 U4_Y 预焊上料Z轴运行条件
LDNOT 812.02  ; RK_12 U4_Y 预焊上料Z轴报警信号标志[0012.02]
AND 812.03  ; RK_12 U4_Y 预焊上料Z轴准备好了信号标志[0012.03]
ANDNOT 200.01  ; 紧急停止
ANDNOT 2042.15  ; RK_12 U4_Y 预焊上料Z轴停止
OUT D1222.02  ; RK_12 U4_Y 预焊上料Z轴运行条件
; rung 43: RK_12 U4_Y 预焊上料Z轴回原点条件
LD P_On
OUT D1222.03  ; RK_12 U4_Y 预焊上料Z轴回原点条件

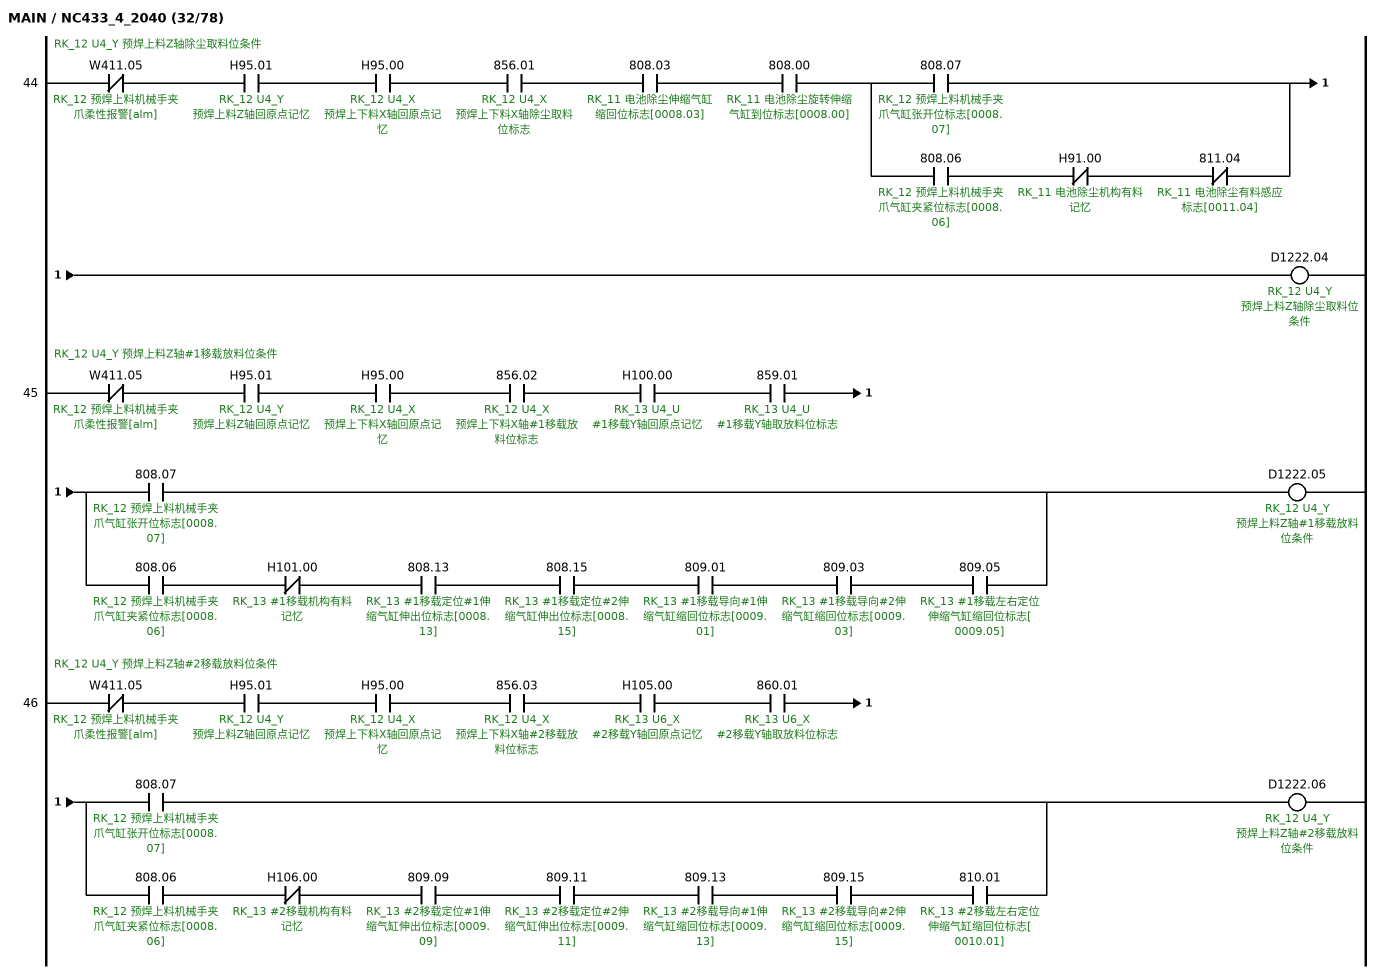
; rung 44: RK_12 U4_Y 预焊上料Z轴除尘取料位条件
LDNOT W411.05  ; RK_12 预焊上料机械手夹爪柔性报警[alm]
AND H95.01  ; RK_12 U4_Y 预焊上料Z轴回原点记忆
AND H95.00  ; RK_12 U4_X 预焊上下料X轴回原点记忆
AND 856.01  ; RK_12 U4_X 预焊上下料X轴除尘取料位标志
AND 808.03  ; RK_11 电池除尘伸缩气缸缩回位标志[0008.03]
AND 808.00  ; RK_11 电池除尘旋转伸缩气缸到位标志[0008.00]
LD 808.07  ; RK_12 预焊上料机械手夹爪气缸张开位标志[0008.07]
LD 808.06  ; RK_12 预焊上料机械手夹爪气缸夹紧位标志[0008.06]
ANDNOT H91.00  ; RK_11 电池除尘机构有料记忆
ANDNOT 811.04  ; RK_11 电池除尘有料感应标志[0011.04]
ORLD
ANDLD
OUT D1222.04  ; RK_12 U4_Y 预焊上料Z轴除尘取料位条件
; rung 45: RK_12 U4_Y 预焊上料Z轴#1移载放料位条件
LDNOT W411.05  ; RK_12 预焊上料机械手夹爪柔性报警[alm]
AND H95.01  ; RK_12 U4_Y 预焊上料Z轴回原点记忆
AND H95.00  ; RK_12 U4_X 预焊上下料X轴回原点记忆
AND 856.02  ; RK_12 U4_X 预焊上下料X轴#1移载放料位标志
AND H100.00  ; RK_13 U4_U #1移载Y轴回原点记忆
AND 859.01  ; RK_13 U4_U #1移载Y轴取放料位标志
LD 808.07  ; RK_12 预焊上料机械手夹爪气缸张开位标志[0008.07]
LD 808.06  ; RK_12 预焊上料机械手夹爪气缸夹紧位标志[0008.06]
ANDNOT H101.00  ; RK_13 #1移载机构有料记忆
AND 808.13  ; RK_13 #1移载定位#1伸缩气缸伸出位标志[0008.13]
AND 808.15  ; RK_13 #1移载定位#2伸缩气缸伸出位标志[0008.15]
AND 809.01  ; RK_13 #1移载导向#1伸缩气缸缩回位标志[0009.01]
AND 809.03  ; RK_13 #1移载导向#2伸缩气缸缩回位标志[0009.03]
AND 809.05  ; RK_13 #1移载左右定位伸缩气缸缩回位标志[0009.05]
ORLD
ANDLD
OUT D1222.05  ; RK_12 U4_Y 预焊上料Z轴#1移载放料位条件
; rung 46: RK_12 U4_Y 预焊上料Z轴#2移载放料位条件
LDNOT W411.05  ; RK_12 预焊上料机械手夹爪柔性报警[alm]
AND H95.01  ; RK_12 U4_Y 预焊上料Z轴回原点记忆
AND H95.00  ; RK_12 U4_X 预焊上下料X轴回原点记忆
AND 856.03  ; RK_12 U4_X 预焊上下料X轴#2移载放料位标志
AND H105.00  ; RK_13 U6_X #2移载Y轴回原点记忆
AND 860.01  ; RK_13 U6_X #2移载Y轴取放料位标志
LD 808.07  ; RK_12 预焊上料机械手夹爪气缸张开位标志[0008.07]
LD 808.06  ; RK_12 预焊上料机械手夹爪气缸夹紧位标志[0008.06]
ANDNOT H106.00  ; RK_13 #2移载机构有料记忆
AND 809.09  ; RK_13 #2移载定位#1伸缩气缸伸出位标志[0009.09]
AND 809.11  ; RK_13 #2移载定位#2伸缩气缸伸出位标志[0009.11]
AND 809.13  ; RK_13 #2移载导向#1伸缩气缸缩回位标志[0009.13]
AND 809.15  ; RK_13 #2移载导向#2伸缩气缸缩回位标志[0009.15]
AND 810.01  ; RK_13 #2移载左右定位伸缩气缸缩回位标志[0010.01]
ORLD
ANDLD
OUT D1222.06  ; RK_12 U4_Y 预焊上料Z轴#2移载放料位条件

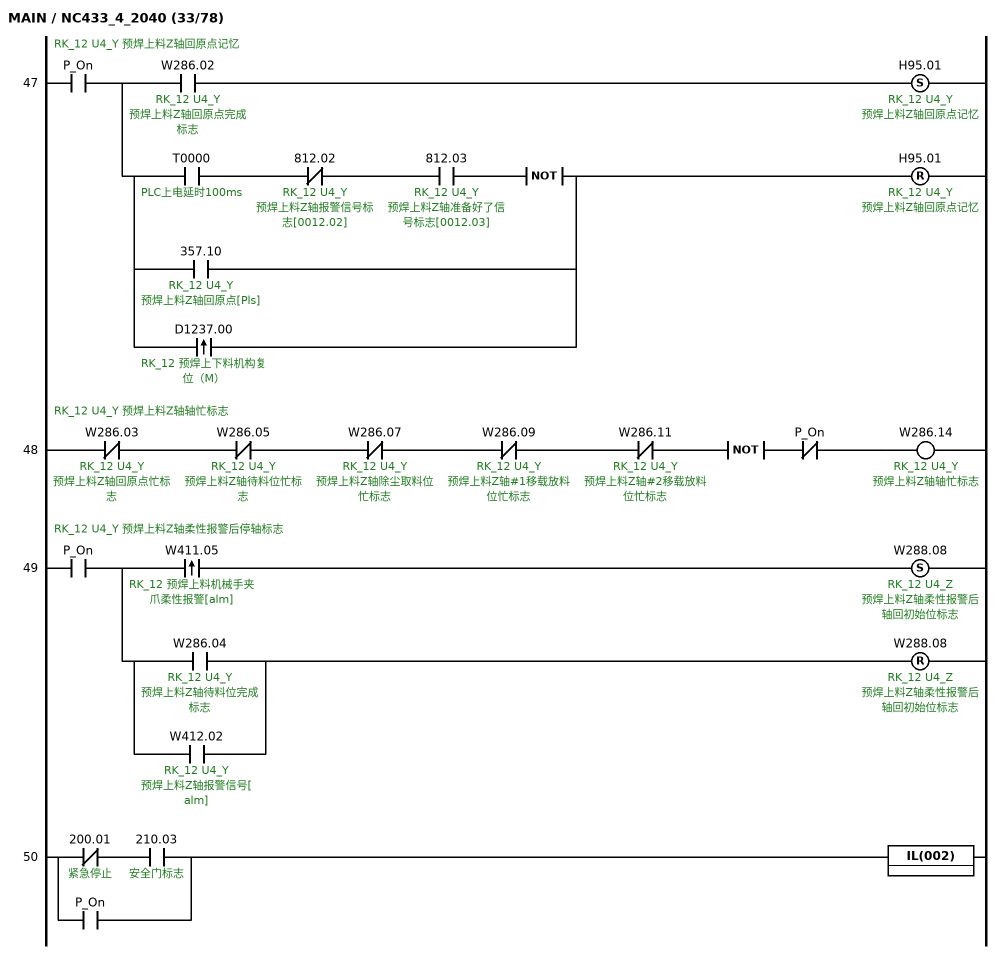
; rung 47: RK_12 U4_Y 预焊上料Z轴回原点记忆
LD P_On
OUT TR0
AND W286.02  ; RK_12 U4_Y 预焊上料Z轴回原点完成标志
SET H95.01  ; RK_12 U4_Y 预焊上料Z轴回原点记忆
LD TR0
LD T0000  ; PLC上电延时100ms
ANDNOT 812.02  ; RK_12 U4_Y 预焊上料Z轴报警信号标志[0012.02]
AND 812.03  ; RK_12 U4_Y 预焊上料Z轴准备好了信号标志[0012.03]
NOT(520)
OR 357.10  ; RK_12 U4_Y 预焊上料Z轴回原点[Pls]
@OR D1237.00  ; RK_12 预焊上下料机构复位（M）
ANDLD
RSET H95.01  ; RK_12 U4_Y 预焊上料Z轴回原点记忆
; rung 48: RK_12 U4_Y 预焊上料Z轴轴忙标志
LDNOT W286.03  ; RK_12 U4_Y 预焊上料Z轴回原点忙标志
ANDNOT W286.05  ; RK_12 U4_Y 预焊上料Z轴待料位忙标志
ANDNOT W286.07  ; RK_12 U4_Y 预焊上料Z轴除尘取料位忙标志
ANDNOT W286.09  ; RK_12 U4_Y 预焊上料Z轴#1移载放料位忙标志
ANDNOT W286.11  ; RK_12 U4_Y 预焊上料Z轴#2移载放料位忙标志
NOT(520)
ANDNOT P_On
OUT W286.14  ; RK_12 U4_Y 预焊上料Z轴轴忙标志
; rung 49: RK_12 U4_Y 预焊上料Z轴柔性报警后停轴标志
LD P_On
OUT TR0
@AND W411.05  ; RK_12 预焊上料机械手夹爪柔性报警[alm]
SET W288.08  ; RK_12 U4_Z 预焊上料Z轴柔性报警后轴回初始位标志
LD TR0
LD W286.04  ; RK_12 U4_Y 预焊上料Z轴待料位完成标志
OR W412.02  ; RK_12 U4_Y 预焊上料Z轴报警信号[alm]
ANDLD
RSET W288.08  ; RK_12 U4_Z 预焊上料Z轴柔性报警后轴回初始位标志
; rung 50
LDNOT 200.01  ; 紧急停止
AND 210.03  ; 安全门标志
OR P_On
IL(002)

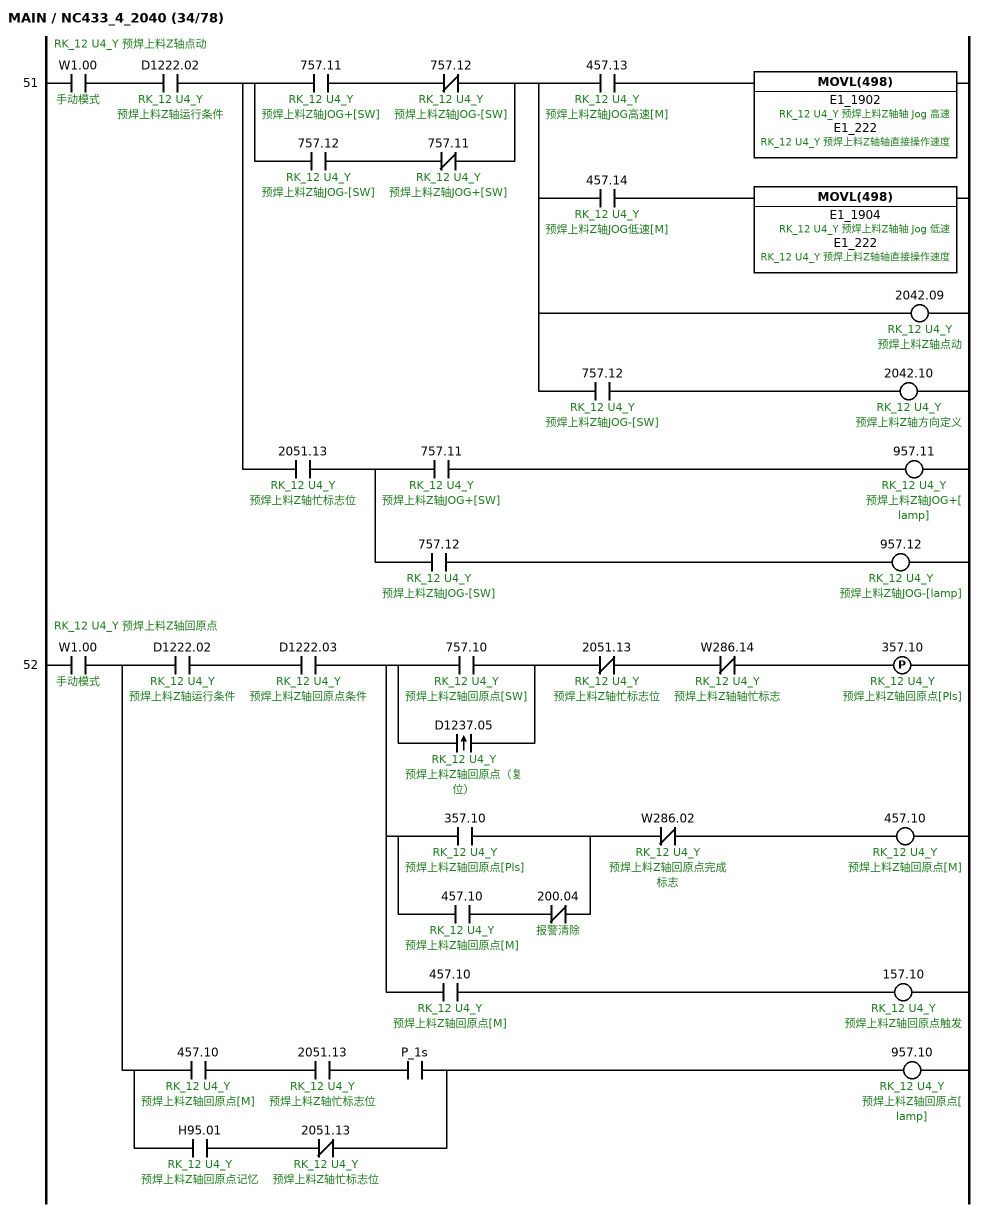
; rung 51: RK_12 U4_Y 预焊上料Z轴点动
LD W1.00  ; 手动模式
AND D1222.02  ; RK_12 U4_Y 预焊上料Z轴运行条件
OUT TR0
LD 757.11  ; RK_12 U4_Y 预焊上料Z轴JOG+[SW]
ANDNOT 757.12  ; RK_12 U4_Y 预焊上料Z轴JOG-[SW]
LD 757.12  ; RK_12 U4_Y 预焊上料Z轴JOG-[SW]
ANDNOT 757.11  ; RK_12 U4_Y 预焊上料Z轴JOG+[SW]
ORLD
ANDLD
OUT TR1
AND 457.13  ; RK_12 U4_Y 预焊上料Z轴JOG高速[M]
MOVL(498) E1_1902 E1_222  ; RK_12 U4_Y 预焊上料Z轴轴 Jog 高速, RK_12 U4_Y 预焊上料Z轴轴直接操作速度
LD TR1
AND 457.14  ; RK_12 U4_Y 预焊上料Z轴JOG低速[M]
MOVL(498) E1_1904 E1_222  ; RK_12 U4_Y 预焊上料Z轴轴 Jog 低速, RK_12 U4_Y 预焊上料Z轴轴直接操作速度
LD TR1
OUT 2042.09  ; RK_12 U4_Y 预焊上料Z轴点动
AND 757.12  ; RK_12 U4_Y 预焊上料Z轴JOG-[SW]
OUT 2042.10  ; RK_12 U4_Y 预焊上料Z轴方向定义
LD TR0
AND 2051.13  ; RK_12 U4_Y 预焊上料Z轴忙标志位
OUT TR0
AND 757.11  ; RK_12 U4_Y 预焊上料Z轴JOG+[SW]
OUT 957.11  ; RK_12 U4_Y 预焊上料Z轴JOG+[lamp]
LD TR0
AND 757.12  ; RK_12 U4_Y 预焊上料Z轴JOG-[SW]
OUT 957.12  ; RK_12 U4_Y 预焊上料Z轴JOG-[lamp]
; rung 52: RK_12 U4_Y 预焊上料Z轴回原点
LD W1.00  ; 手动模式
OUT TR0
AND D1222.02  ; RK_12 U4_Y 预焊上料Z轴运行条件
AND D1222.03  ; RK_12 U4_Y 预焊上料Z轴回原点条件
OUT TR1
LD 757.10  ; RK_12 U4_Y 预焊上料Z轴回原点[SW]
@OR D1237.05  ; RK_12 U4_Y 预焊上料Z轴回原点（复位）
ANDLD
ANDNOT 2051.13  ; RK_12 U4_Y 预焊上料Z轴忙标志位
ANDNOT W286.14  ; RK_12 U4_Y 预焊上料Z轴轴忙标志
DIFU(013) 357.10  ; RK_12 U4_Y 预焊上料Z轴回原点[Pls]
LD TR1
LD 357.10  ; RK_12 U4_Y 预焊上料Z轴回原点[Pls]
LD 457.10  ; RK_12 U4_Y 预焊上料Z轴回原点[M]
ANDNOT 200.04  ; 报警清除
ORLD
ANDLD
ANDNOT W286.02  ; RK_12 U4_Y 预焊上料Z轴回原点完成标志
OUT 457.10  ; RK_12 U4_Y 预焊上料Z轴回原点[M]
LD TR1
AND 457.10  ; RK_12 U4_Y 预焊上料Z轴回原点[M]
OUT 157.10  ; RK_12 U4_Y 预焊上料Z轴回原点触发
LD TR0
LD 457.10  ; RK_12 U4_Y 预焊上料Z轴回原点[M]
AND 2051.13  ; RK_12 U4_Y 预焊上料Z轴忙标志位
AND P_1s
LD H95.01  ; RK_12 U4_Y 预焊上料Z轴回原点记忆
ANDNOT 2051.13  ; RK_12 U4_Y 预焊上料Z轴忙标志位
ORLD
ANDLD
OUT 957.10  ; RK_12 U4_Y 预焊上料Z轴回原点[lamp]

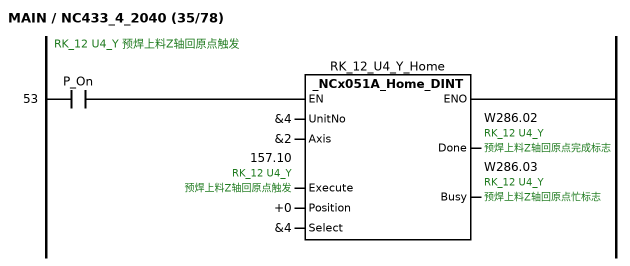
; rung 53: RK_12 U4_Y 预焊上料Z轴回原点触发
LD P_On
CALL RK_12_U4_Y_Home : _NCx051A_Home_DINT (UnitNo := &4, Axis := &2, Execute := 157.10, Position := +0, Select := &4, Done => W286.02, Busy => W286.03)  ; RK_12 U4_Y 预焊上料Z轴回原点触发, RK_12 U4_Y 预焊上料Z轴回原点完成标志, RK_12 U4_Y 预焊上料Z轴回原点忙标志

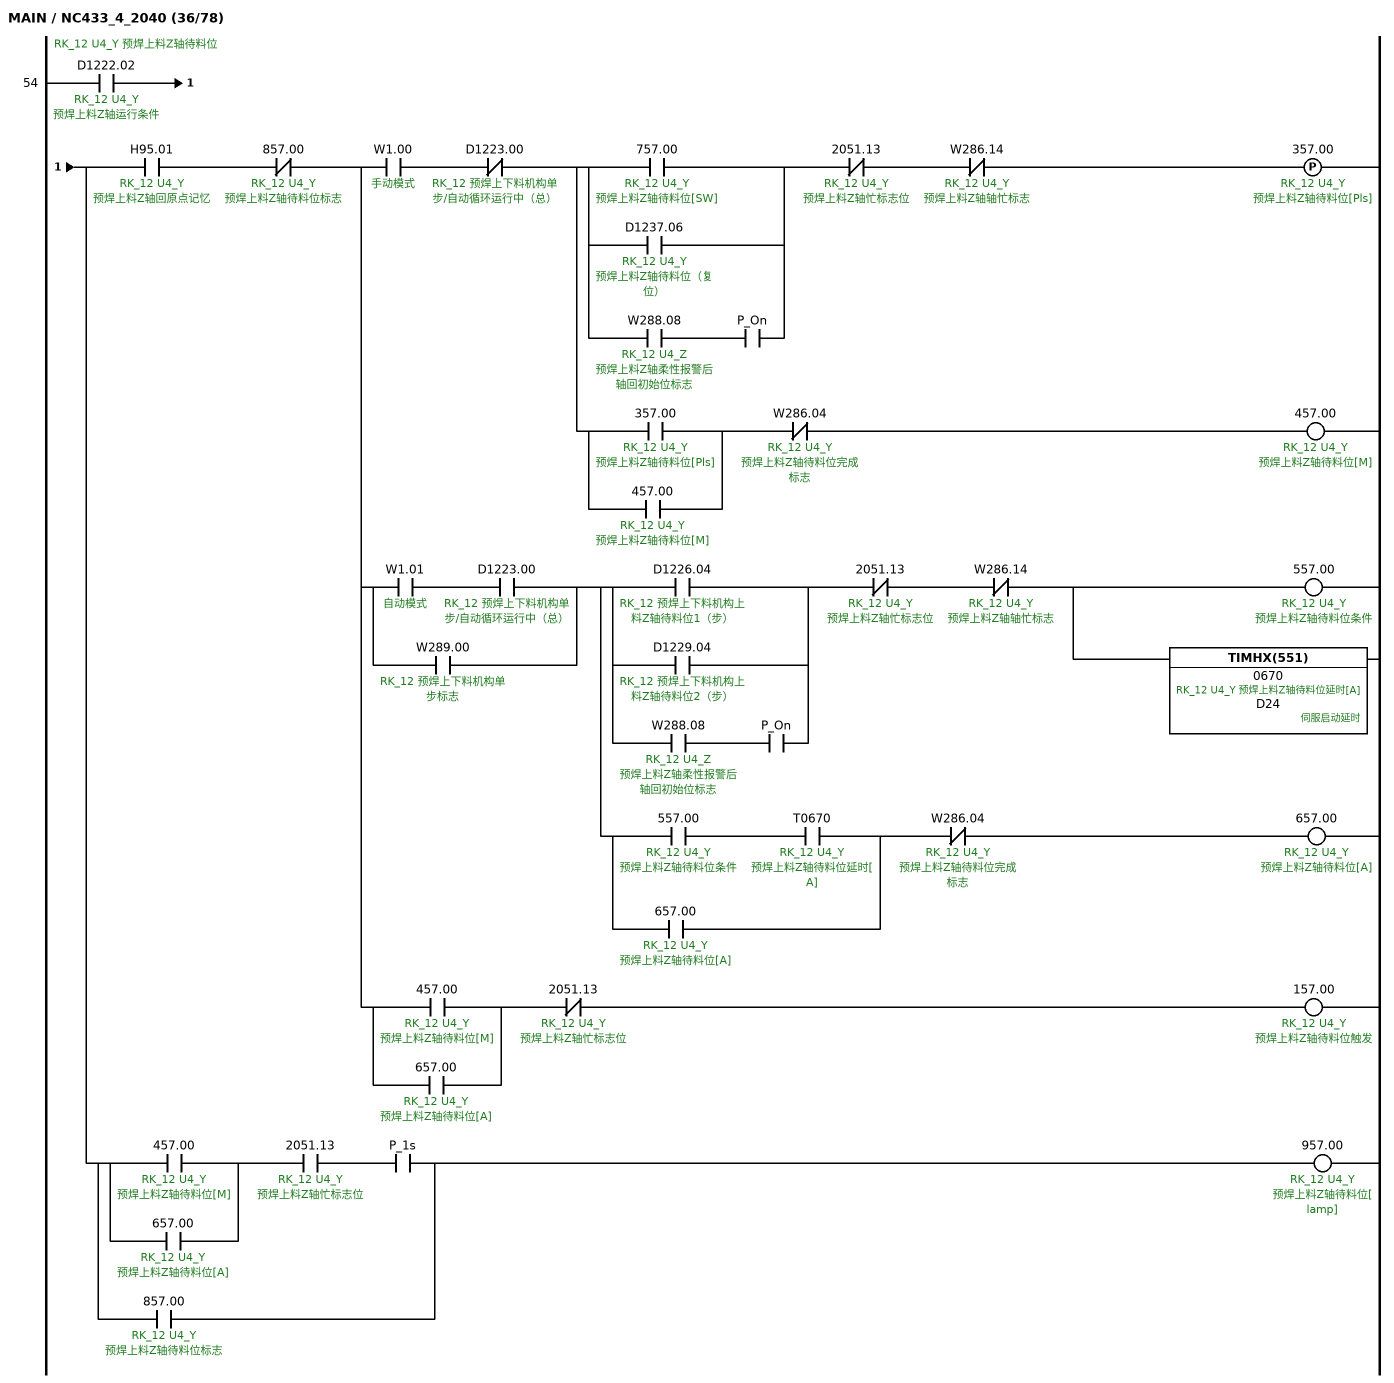
; rung 54: RK_12 U4_Y 预焊上料Z轴待料位
LD D1222.02  ; RK_12 U4_Y 预焊上料Z轴运行条件
OUT TR0
AND H95.01  ; RK_12 U4_Y 预焊上料Z轴回原点记忆
ANDNOT 857.00  ; RK_12 U4_Y 预焊上料Z轴待料位标志
OUT TR1
AND W1.00  ; 手动模式
ANDNOT D1223.00  ; RK_12 预焊上下料机构单步/自动循环运行中（总）
OUT TR2
LD 757.00  ; RK_12 U4_Y 预焊上料Z轴待料位[SW]
OR D1237.06  ; RK_12 U4_Y 预焊上料Z轴待料位（复位）
LD W288.08  ; RK_12 U4_Z 预焊上料Z轴柔性报警后轴回初始位标志
AND P_On
ORLD
ANDLD
ANDNOT 2051.13  ; RK_12 U4_Y 预焊上料Z轴忙标志位
ANDNOT W286.14  ; RK_12 U4_Y 预焊上料Z轴轴忙标志
DIFU(013) 357.00  ; RK_12 U4_Y 预焊上料Z轴待料位[Pls]
LD TR2
LD 357.00  ; RK_12 U4_Y 预焊上料Z轴待料位[Pls]
OR 457.00  ; RK_12 U4_Y 预焊上料Z轴待料位[M]
ANDLD
ANDNOT W286.04  ; RK_12 U4_Y 预焊上料Z轴待料位完成标志
OUT 457.00  ; RK_12 U4_Y 预焊上料Z轴待料位[M]
LD TR1
LD W1.01  ; 自动模式
AND D1223.00  ; RK_12 预焊上下料机构单步/自动循环运行中（总）
OR W289.00  ; RK_12 预焊上下料机构单步标志
ANDLD
OUT TR2
LD D1226.04  ; RK_12 预焊上下料机构上料Z轴待料位1（步）
OR D1229.04  ; RK_12 预焊上下料机构上料Z轴待料位2（步）
LD W288.08  ; RK_12 U4_Z 预焊上料Z轴柔性报警后轴回初始位标志
AND P_On
ORLD
ANDLD
ANDNOT 2051.13  ; RK_12 U4_Y 预焊上料Z轴忙标志位
ANDNOT W286.14  ; RK_12 U4_Y 预焊上料Z轴轴忙标志
OUT 557.00  ; RK_12 U4_Y 预焊上料Z轴待料位条件
TIMHX(551) 0670 D24  ; 伺服启动延时, RK_12 U4_Y 预焊上料Z轴待料位延时[A]
LD TR2
LD 557.00  ; RK_12 U4_Y 预焊上料Z轴待料位条件
AND T0670  ; RK_12 U4_Y 预焊上料Z轴待料位延时[A]
OR 657.00  ; RK_12 U4_Y 预焊上料Z轴待料位[A]
ANDLD
ANDNOT W286.04  ; RK_12 U4_Y 预焊上料Z轴待料位完成标志
OUT 657.00  ; RK_12 U4_Y 预焊上料Z轴待料位[A]
LD TR1
LD 457.00  ; RK_12 U4_Y 预焊上料Z轴待料位[M]
OR 657.00  ; RK_12 U4_Y 预焊上料Z轴待料位[A]
ANDLD
ANDNOT 2051.13  ; RK_12 U4_Y 预焊上料Z轴忙标志位
OUT 157.00  ; RK_12 U4_Y 预焊上料Z轴待料位触发
LD TR0
LD 457.00  ; RK_12 U4_Y 预焊上料Z轴待料位[M]
OR 657.00  ; RK_12 U4_Y 预焊上料Z轴待料位[A]
AND 2051.13  ; RK_12 U4_Y 预焊上料Z轴忙标志位
AND P_1s
OR 857.00  ; RK_12 U4_Y 预焊上料Z轴待料位标志
ANDLD
OUT 957.00  ; RK_12 U4_Y 预焊上料Z轴待料位[lamp]

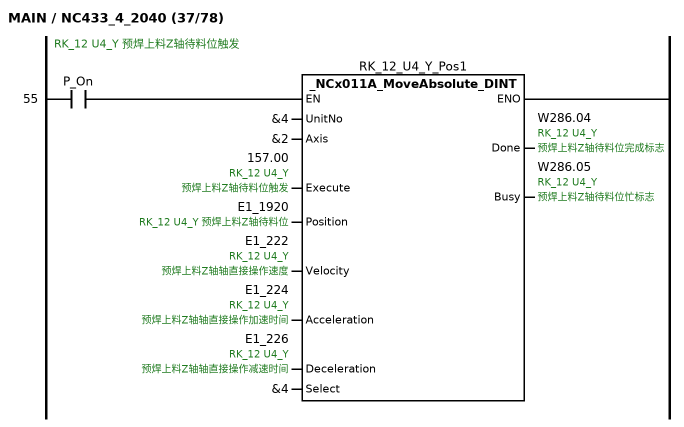
; rung 55: RK_12 U4_Y 预焊上料Z轴待料位触发
LD P_On
CALL RK_12_U4_Y_Pos1 : _NCx011A_MoveAbsolute_DINT (UnitNo := &4, Axis := &2, Execute := 157.00, Position := E1_1920, Velocity := E1_222, Acceleration := E1_224, Deceleration := E1_226, Select := &4, Done => W286.04, Busy => W286.05)  ; RK_12 U4_Y 预焊上料Z轴待料位触发, RK_12 U4_Y 预焊上料Z轴待料位, RK_12 U4_Y 预焊上料Z轴轴直接操作速度, RK_12 U4_Y 预焊上料Z轴轴直接操作加速时间, RK_12 U4_Y 预焊上料Z轴轴直接操作减速时间, RK_12 U4_Y 预焊上料Z轴待料位完成标志, RK_12 U4_Y 预焊上料Z轴待料位忙标志

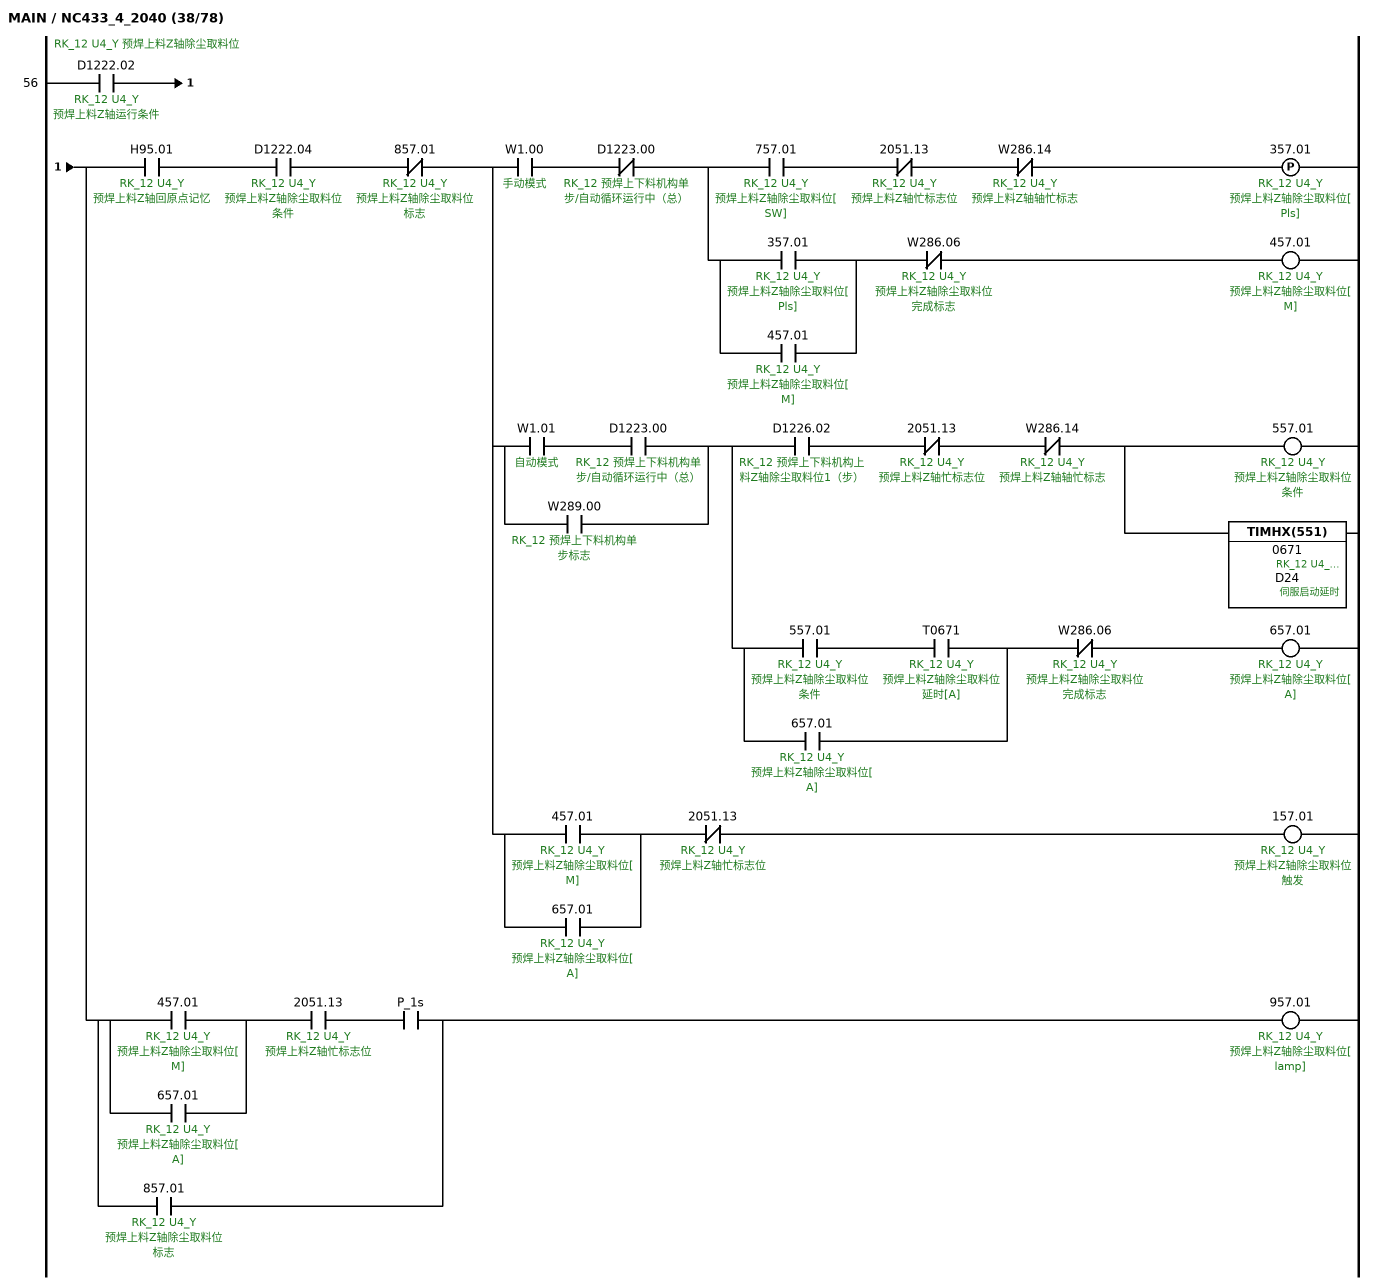
; rung 56: RK_12 U4_Y 预焊上料Z轴除尘取料位
LD D1222.02  ; RK_12 U4_Y 预焊上料Z轴运行条件
OUT TR0
AND H95.01  ; RK_12 U4_Y 预焊上料Z轴回原点记忆
AND D1222.04  ; RK_12 U4_Y 预焊上料Z轴除尘取料位条件
ANDNOT 857.01  ; RK_12 U4_Y 预焊上料Z轴除尘取料位标志
OUT TR1
AND W1.00  ; 手动模式
ANDNOT D1223.00  ; RK_12 预焊上下料机构单步/自动循环运行中（总）
OUT TR2
AND 757.01  ; RK_12 U4_Y 预焊上料Z轴除尘取料位[SW]
ANDNOT 2051.13  ; RK_12 U4_Y 预焊上料Z轴忙标志位
ANDNOT W286.14  ; RK_12 U4_Y 预焊上料Z轴轴忙标志
DIFU(013) 357.01  ; RK_12 U4_Y 预焊上料Z轴除尘取料位[Pls]
LD TR2
LD 357.01  ; RK_12 U4_Y 预焊上料Z轴除尘取料位[Pls]
OR 457.01  ; RK_12 U4_Y 预焊上料Z轴除尘取料位[M]
ANDLD
ANDNOT W286.06  ; RK_12 U4_Y 预焊上料Z轴除尘取料位完成标志
OUT 457.01  ; RK_12 U4_Y 预焊上料Z轴除尘取料位[M]
LD TR1
LD W1.01  ; 自动模式
AND D1223.00  ; RK_12 预焊上下料机构单步/自动循环运行中（总）
OR W289.00  ; RK_12 预焊上下料机构单步标志
ANDLD
OUT TR2
AND D1226.02  ; RK_12 预焊上下料机构上料Z轴除尘取料位1（步）
ANDNOT 2051.13  ; RK_12 U4_Y 预焊上料Z轴忙标志位
ANDNOT W286.14  ; RK_12 U4_Y 预焊上料Z轴轴忙标志
OUT 557.01  ; RK_12 U4_Y 预焊上料Z轴除尘取料位条件
TIMHX(551) 0671 D24  ; 伺服启动延时, RK_12 U4_Y 预焊上料Z轴除尘取料位延时[A]
LD TR2
LD 557.01  ; RK_12 U4_Y 预焊上料Z轴除尘取料位条件
AND T0671  ; RK_12 U4_Y 预焊上料Z轴除尘取料位延时[A]
OR 657.01  ; RK_12 U4_Y 预焊上料Z轴除尘取料位[A]
ANDLD
ANDNOT W286.06  ; RK_12 U4_Y 预焊上料Z轴除尘取料位完成标志
OUT 657.01  ; RK_12 U4_Y 预焊上料Z轴除尘取料位[A]
LD TR1
LD 457.01  ; RK_12 U4_Y 预焊上料Z轴除尘取料位[M]
OR 657.01  ; RK_12 U4_Y 预焊上料Z轴除尘取料位[A]
ANDLD
ANDNOT 2051.13  ; RK_12 U4_Y 预焊上料Z轴忙标志位
OUT 157.01  ; RK_12 U4_Y 预焊上料Z轴除尘取料位触发
LD TR0
LD 457.01  ; RK_12 U4_Y 预焊上料Z轴除尘取料位[M]
OR 657.01  ; RK_12 U4_Y 预焊上料Z轴除尘取料位[A]
AND 2051.13  ; RK_12 U4_Y 预焊上料Z轴忙标志位
AND P_1s
OR 857.01  ; RK_12 U4_Y 预焊上料Z轴除尘取料位标志
ANDLD
OUT 957.01  ; RK_12 U4_Y 预焊上料Z轴除尘取料位[lamp]

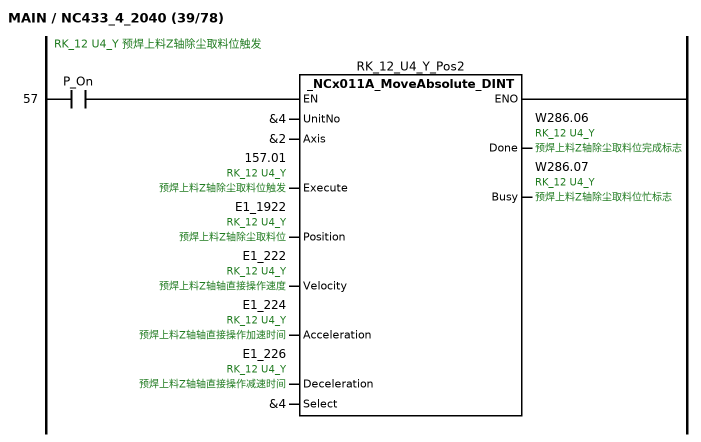
; rung 57: RK_12 U4_Y 预焊上料Z轴除尘取料位触发
LD P_On
CALL RK_12_U4_Y_Pos2 : _NCx011A_MoveAbsolute_DINT (UnitNo := &4, Axis := &2, Execute := 157.01, Position := E1_1922, Velocity := E1_222, Acceleration := E1_224, Deceleration := E1_226, Select := &4, Done => W286.06, Busy => W286.07)  ; RK_12 U4_Y 预焊上料Z轴除尘取料位触发, RK_12 U4_Y 预焊上料Z轴除尘取料位, RK_12 U4_Y 预焊上料Z轴轴直接操作速度, RK_12 U4_Y 预焊上料Z轴轴直接操作加速时间, RK_12 U4_Y 预焊上料Z轴轴直接操作减速时间, RK_12 U4_Y 预焊上料Z轴除尘取料位完成标志, RK_12 U4_Y 预焊上料Z轴除尘取料位忙标志

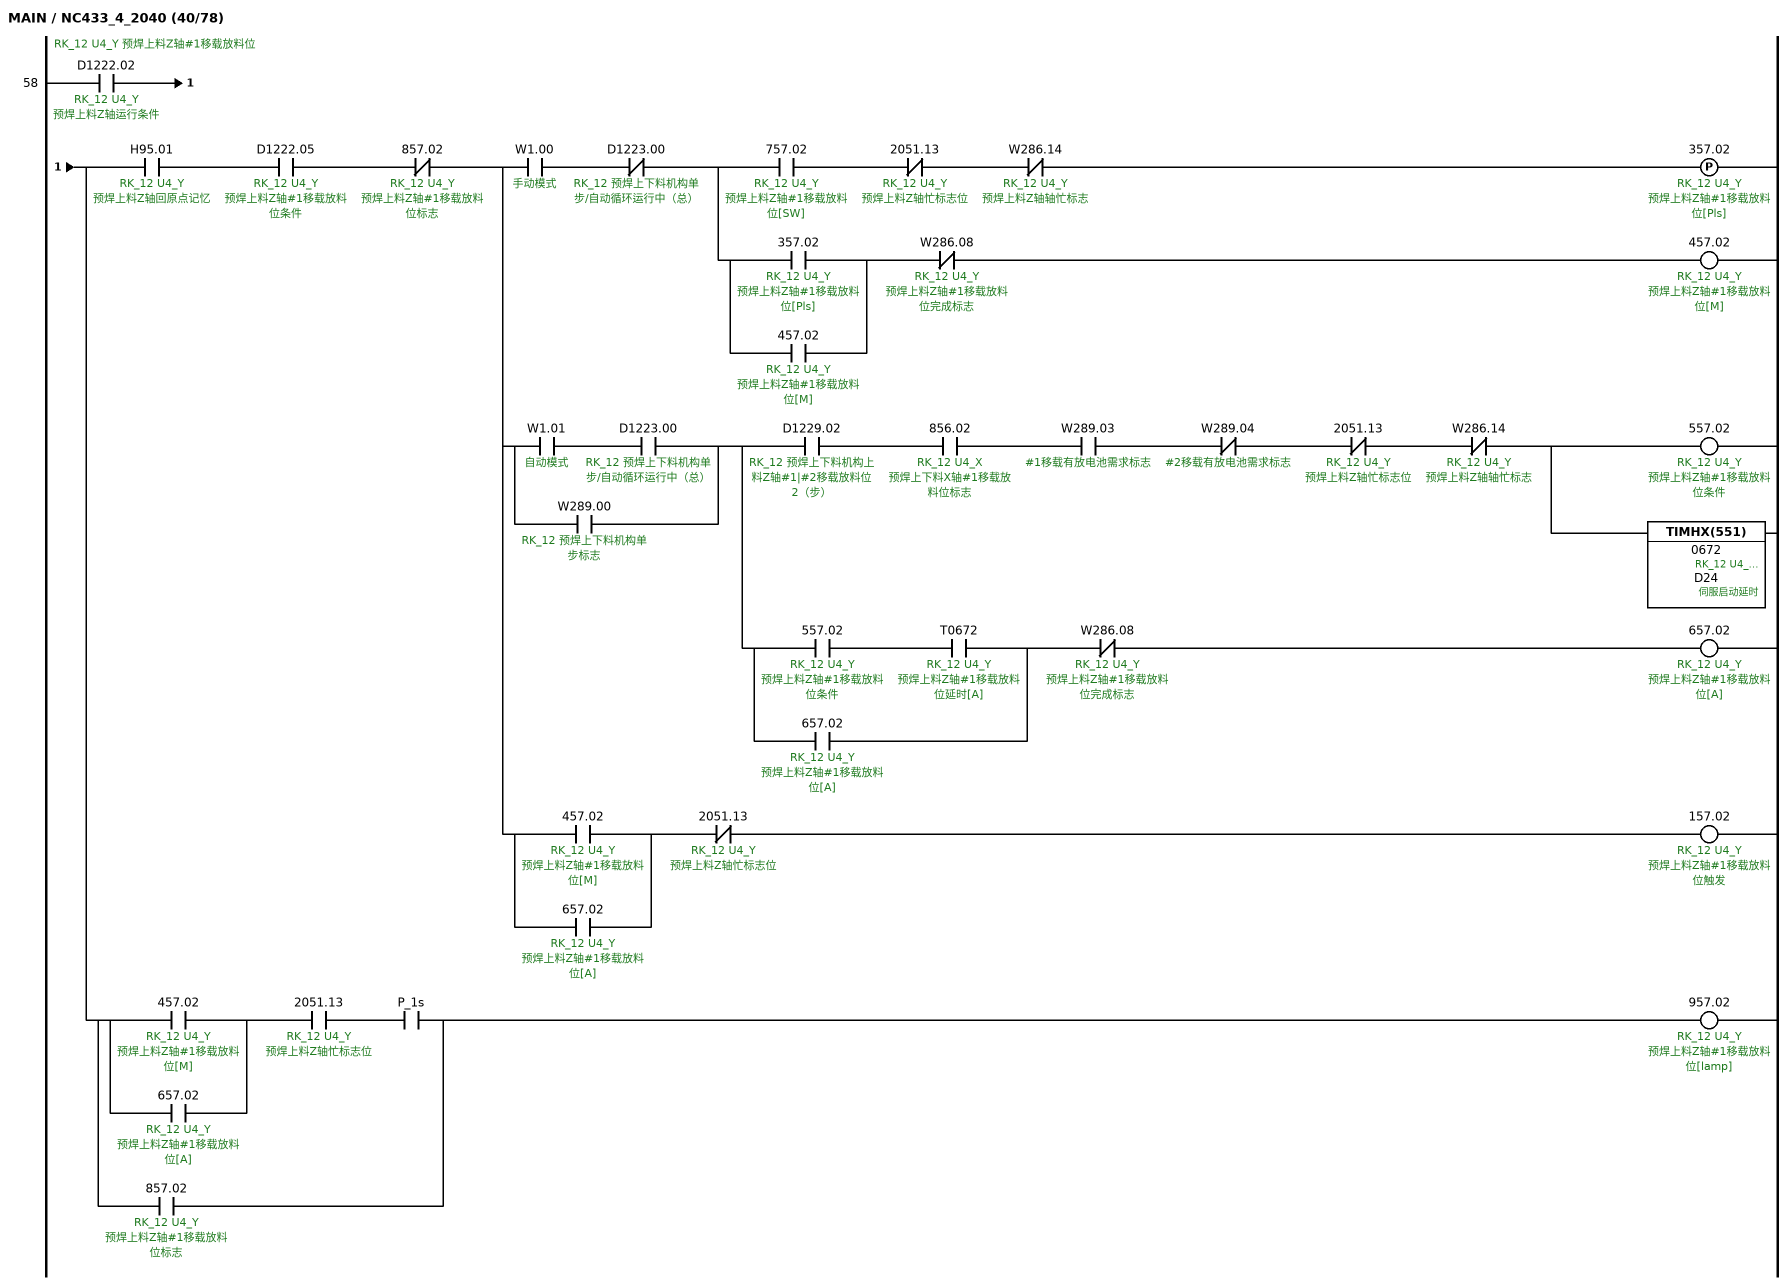
; rung 58: RK_12 U4_Y 预焊上料Z轴#1移载放料位
LD D1222.02  ; RK_12 U4_Y 预焊上料Z轴运行条件
OUT TR0
AND H95.01  ; RK_12 U4_Y 预焊上料Z轴回原点记忆
AND D1222.05  ; RK_12 U4_Y 预焊上料Z轴#1移载放料位条件
ANDNOT 857.02  ; RK_12 U4_Y 预焊上料Z轴#1移载放料位标志
OUT TR1
AND W1.00  ; 手动模式
ANDNOT D1223.00  ; RK_12 预焊上下料机构单步/自动循环运行中（总）
OUT TR2
AND 757.02  ; RK_12 U4_Y 预焊上料Z轴#1移载放料位[SW]
ANDNOT 2051.13  ; RK_12 U4_Y 预焊上料Z轴忙标志位
ANDNOT W286.14  ; RK_12 U4_Y 预焊上料Z轴轴忙标志
DIFU(013) 357.02  ; RK_12 U4_Y 预焊上料Z轴#1移载放料位[Pls]
LD TR2
LD 357.02  ; RK_12 U4_Y 预焊上料Z轴#1移载放料位[Pls]
OR 457.02  ; RK_12 U4_Y 预焊上料Z轴#1移载放料位[M]
ANDLD
ANDNOT W286.08  ; RK_12 U4_Y 预焊上料Z轴#1移载放料位完成标志
OUT 457.02  ; RK_12 U4_Y 预焊上料Z轴#1移载放料位[M]
LD TR1
LD W1.01  ; 自动模式
AND D1223.00  ; RK_12 预焊上下料机构单步/自动循环运行中（总）
OR W289.00  ; RK_12 预焊上下料机构单步标志
ANDLD
OUT TR2
AND D1229.02  ; RK_12 预焊上下料机构上料Z轴#1|#2移载放料位2（步）
AND 856.02  ; RK_12 U4_X 预焊上下料X轴#1移载放料位标志
AND W289.03  ; #1移载有放电池需求标志
ANDNOT W289.04  ; #2移载有放电池需求标志
ANDNOT 2051.13  ; RK_12 U4_Y 预焊上料Z轴忙标志位
ANDNOT W286.14  ; RK_12 U4_Y 预焊上料Z轴轴忙标志
OUT 557.02  ; RK_12 U4_Y 预焊上料Z轴#1移载放料位条件
TIMHX(551) 0672 D24  ; 伺服启动延时, RK_12 U4_Y 预焊上料Z轴#1移载放料位延时[A]
LD TR2
LD 557.02  ; RK_12 U4_Y 预焊上料Z轴#1移载放料位条件
AND T0672  ; RK_12 U4_Y 预焊上料Z轴#1移载放料位延时[A]
OR 657.02  ; RK_12 U4_Y 预焊上料Z轴#1移载放料位[A]
ANDLD
ANDNOT W286.08  ; RK_12 U4_Y 预焊上料Z轴#1移载放料位完成标志
OUT 657.02  ; RK_12 U4_Y 预焊上料Z轴#1移载放料位[A]
LD TR1
LD 457.02  ; RK_12 U4_Y 预焊上料Z轴#1移载放料位[M]
OR 657.02  ; RK_12 U4_Y 预焊上料Z轴#1移载放料位[A]
ANDLD
ANDNOT 2051.13  ; RK_12 U4_Y 预焊上料Z轴忙标志位
OUT 157.02  ; RK_12 U4_Y 预焊上料Z轴#1移载放料位触发
LD TR0
LD 457.02  ; RK_12 U4_Y 预焊上料Z轴#1移载放料位[M]
OR 657.02  ; RK_12 U4_Y 预焊上料Z轴#1移载放料位[A]
AND 2051.13  ; RK_12 U4_Y 预焊上料Z轴忙标志位
AND P_1s
OR 857.02  ; RK_12 U4_Y 预焊上料Z轴#1移载放料位标志
ANDLD
OUT 957.02  ; RK_12 U4_Y 预焊上料Z轴#1移载放料位[lamp]

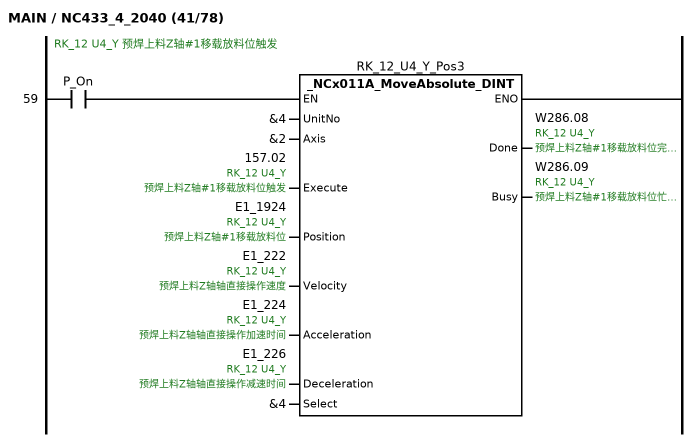
; rung 59: RK_12 U4_Y 预焊上料Z轴#1移载放料位触发
LD P_On
CALL RK_12_U4_Y_Pos3 : _NCx011A_MoveAbsolute_DINT (UnitNo := &4, Axis := &2, Execute := 157.02, Position := E1_1924, Velocity := E1_222, Acceleration := E1_224, Deceleration := E1_226, Select := &4, Done => W286.08, Busy => W286.09)  ; RK_12 U4_Y 预焊上料Z轴#1移载放料位触发, RK_12 U4_Y 预焊上料Z轴#1移载放料位, RK_12 U4_Y 预焊上料Z轴轴直接操作速度, RK_12 U4_Y 预焊上料Z轴轴直接操作加速时间, RK_12 U4_Y 预焊上料Z轴轴直接操作减速时间, RK_12 U4_Y 预焊上料Z轴#1移载放料位完成标志, RK_12 U4_Y 预焊上料Z轴#1移载放料位忙标志

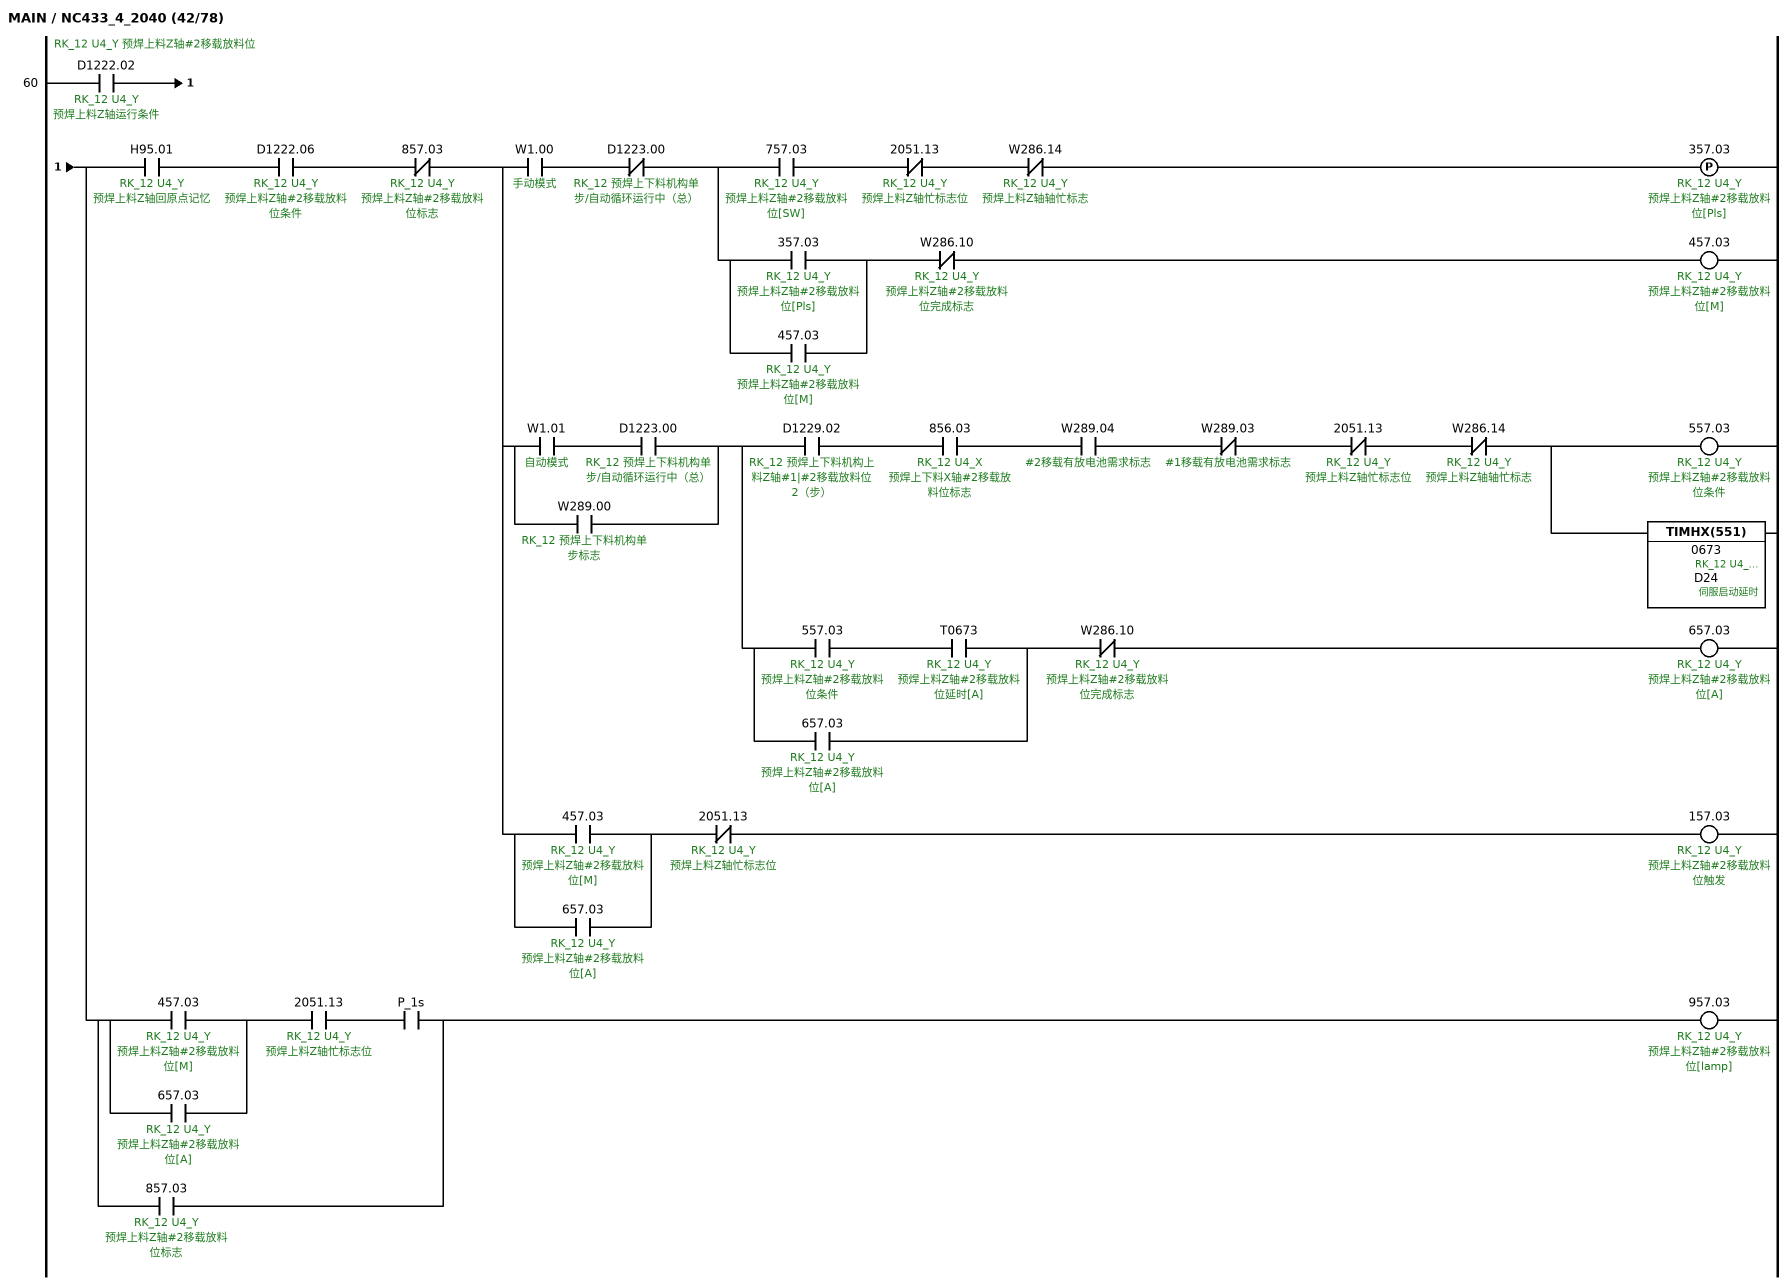
; rung 60: RK_12 U4_Y 预焊上料Z轴#2移载放料位
LD D1222.02  ; RK_12 U4_Y 预焊上料Z轴运行条件
OUT TR0
AND H95.01  ; RK_12 U4_Y 预焊上料Z轴回原点记忆
AND D1222.06  ; RK_12 U4_Y 预焊上料Z轴#2移载放料位条件
ANDNOT 857.03  ; RK_12 U4_Y 预焊上料Z轴#2移载放料位标志
OUT TR1
AND W1.00  ; 手动模式
ANDNOT D1223.00  ; RK_12 预焊上下料机构单步/自动循环运行中（总）
OUT TR2
AND 757.03  ; RK_12 U4_Y 预焊上料Z轴#2移载放料位[SW]
ANDNOT 2051.13  ; RK_12 U4_Y 预焊上料Z轴忙标志位
ANDNOT W286.14  ; RK_12 U4_Y 预焊上料Z轴轴忙标志
DIFU(013) 357.03  ; RK_12 U4_Y 预焊上料Z轴#2移载放料位[Pls]
LD TR2
LD 357.03  ; RK_12 U4_Y 预焊上料Z轴#2移载放料位[Pls]
OR 457.03  ; RK_12 U4_Y 预焊上料Z轴#2移载放料位[M]
ANDLD
ANDNOT W286.10  ; RK_12 U4_Y 预焊上料Z轴#2移载放料位完成标志
OUT 457.03  ; RK_12 U4_Y 预焊上料Z轴#2移载放料位[M]
LD TR1
LD W1.01  ; 自动模式
AND D1223.00  ; RK_12 预焊上下料机构单步/自动循环运行中（总）
OR W289.00  ; RK_12 预焊上下料机构单步标志
ANDLD
OUT TR2
AND D1229.02  ; RK_12 预焊上下料机构上料Z轴#1|#2移载放料位2（步）
AND 856.03  ; RK_12 U4_X 预焊上下料X轴#2移载放料位标志
AND W289.04  ; #2移载有放电池需求标志
ANDNOT W289.03  ; #1移载有放电池需求标志
ANDNOT 2051.13  ; RK_12 U4_Y 预焊上料Z轴忙标志位
ANDNOT W286.14  ; RK_12 U4_Y 预焊上料Z轴轴忙标志
OUT 557.03  ; RK_12 U4_Y 预焊上料Z轴#2移载放料位条件
TIMHX(551) 0673 D24  ; 伺服启动延时, RK_12 U4_Y 预焊上料Z轴#2移载放料位延时[A]
LD TR2
LD 557.03  ; RK_12 U4_Y 预焊上料Z轴#2移载放料位条件
AND T0673  ; RK_12 U4_Y 预焊上料Z轴#2移载放料位延时[A]
OR 657.03  ; RK_12 U4_Y 预焊上料Z轴#2移载放料位[A]
ANDLD
ANDNOT W286.10  ; RK_12 U4_Y 预焊上料Z轴#2移载放料位完成标志
OUT 657.03  ; RK_12 U4_Y 预焊上料Z轴#2移载放料位[A]
LD TR1
LD 457.03  ; RK_12 U4_Y 预焊上料Z轴#2移载放料位[M]
OR 657.03  ; RK_12 U4_Y 预焊上料Z轴#2移载放料位[A]
ANDLD
ANDNOT 2051.13  ; RK_12 U4_Y 预焊上料Z轴忙标志位
OUT 157.03  ; RK_12 U4_Y 预焊上料Z轴#2移载放料位触发
LD TR0
LD 457.03  ; RK_12 U4_Y 预焊上料Z轴#2移载放料位[M]
OR 657.03  ; RK_12 U4_Y 预焊上料Z轴#2移载放料位[A]
AND 2051.13  ; RK_12 U4_Y 预焊上料Z轴忙标志位
AND P_1s
OR 857.03  ; RK_12 U4_Y 预焊上料Z轴#2移载放料位标志
ANDLD
OUT 957.03  ; RK_12 U4_Y 预焊上料Z轴#2移载放料位[lamp]

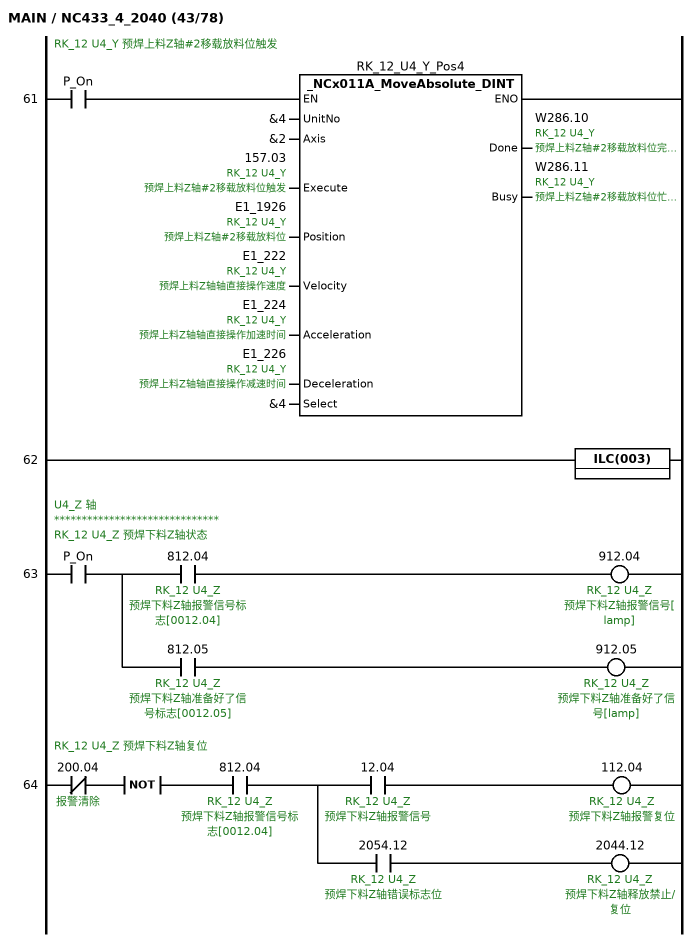
; rung 61: RK_12 U4_Y 预焊上料Z轴#2移载放料位触发
LD P_On
CALL RK_12_U4_Y_Pos4 : _NCx011A_MoveAbsolute_DINT (UnitNo := &4, Axis := &2, Execute := 157.03, Position := E1_1926, Velocity := E1_222, Acceleration := E1_224, Deceleration := E1_226, Select := &4, Done => W286.10, Busy => W286.11)  ; RK_12 U4_Y 预焊上料Z轴#2移载放料位触发, RK_12 U4_Y 预焊上料Z轴#2移载放料位, RK_12 U4_Y 预焊上料Z轴轴直接操作速度, RK_12 U4_Y 预焊上料Z轴轴直接操作加速时间, RK_12 U4_Y 预焊上料Z轴轴直接操作减速时间, RK_12 U4_Y 预焊上料Z轴#2移载放料位完成标志, RK_12 U4_Y 预焊上料Z轴#2移载放料位忙标志
; rung 62
ILC(003)
; rung 63: U4_Z 轴 / ****************************** / RK_12 U4_Z 预焊下料Z轴状态
LD P_On
OUT TR0
AND 812.04  ; RK_12 U4_Z 预焊下料Z轴报警信号标志[0012.04]
OUT 912.04  ; RK_12 U4_Z 预焊下料Z轴报警信号[lamp]
LD TR0
AND 812.05  ; RK_12 U4_Z 预焊下料Z轴准备好了信号标志[0012.05]
OUT 912.05  ; RK_12 U4_Z 预焊下料Z轴准备好了信号[lamp]
; rung 64: RK_12 U4_Z 预焊下料Z轴复位
LDNOT 200.04  ; 报警清除
NOT(520)
AND 812.04  ; RK_12 U4_Z 预焊下料Z轴报警信号标志[0012.04]
OUT TR0
AND 12.04  ; RK_12 U4_Z 预焊下料Z轴报警信号
OUT 112.04  ; RK_12 U4_Z 预焊下料Z轴报警复位
LD TR0
AND 2054.12  ; RK_12 U4_Z 预焊下料Z轴错误标志位
OUT 2044.12  ; RK_12 U4_Z 预焊下料Z轴释放禁止/复位

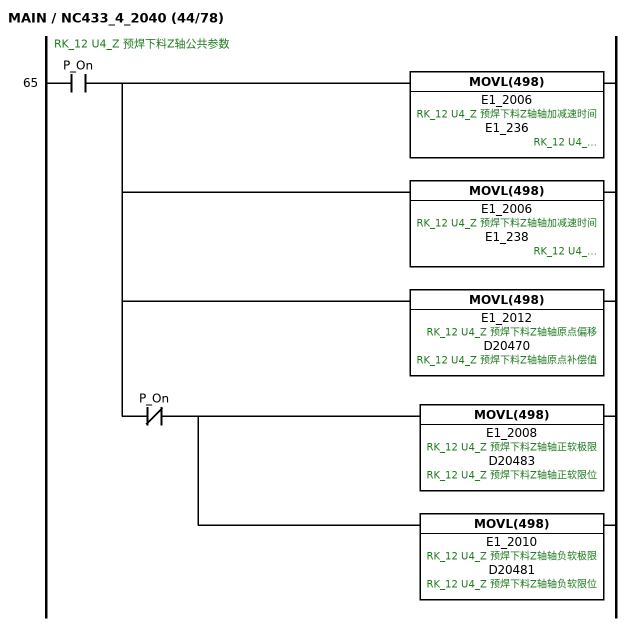
; rung 65: RK_12 U4_Z 预焊下料Z轴公共参数
LD P_On
MOVL(498) E1_2006 E1_236  ; RK_12 U4_Z 预焊下料Z轴轴加减速时间, RK_12 U4_Z 预焊下料Z轴轴直接操作加速时间
MOVL(498) E1_2006 E1_238  ; RK_12 U4_Z 预焊下料Z轴轴加减速时间, RK_12 U4_Z 预焊下料Z轴轴直接操作减速时间
MOVL(498) E1_2012 D20470  ; RK_12 U4_Z 预焊下料Z轴轴原点偏移, RK_12 U4_Z 预焊下料Z轴轴原点补偿值
ANDNOT P_On
MOVL(498) E1_2008 D20483  ; RK_12 U4_Z 预焊下料Z轴轴正软极限, RK_12 U4_Z 预焊下料Z轴轴正软限位
MOVL(498) E1_2010 D20481  ; RK_12 U4_Z 预焊下料Z轴轴负软极限, RK_12 U4_Z 预焊下料Z轴轴负软限位

